// TIA Portal V20 export
FUNCTION_BLOCK "CallUnit"   // FB7, LAD
TITLE = CallUnit
AUTHOR : ERsystem_FA2_DH. Kim
// Unit logic and state machine
// stored: IsIECCheckEnabled true, MemoryReserve 100, Namespace Unit1, SetENOAutomatically false
   VAR_INPUT
      safetyReleased : Bool;   // Status from safety program
   END_VAR
   VAR_OUTPUT
      acknowledgeSafety { ExternalWritable := 'False'} : Bool;   // Acknowledge command to the safety program
   END_VAR
   VAR_IN_OUT
      globalStatus : "LAF_typeGeneralStatus";   // Global status
      unitInterface : "LAF_typeUnitInterface";   // Global unit interface
   END_VAR
   VAR
      instManageAlarms { ExternalWritable := 'False'} : "LAF_ManageAlarms";
      instStatusCollector { ExternalWritable := 'False'} : "LUC_StatusCollector";
      instInterfaceManager { ExternalWritable := 'False'} : "LUC_InterfaceManager";
      instUnitModeStateManager { ExternalWritable := 'False'} : "LPMLV2022_UnitModeStateManager";
      instRemoteInterfaceOpcUa { ExternalWritable := 'False'} : "LUC_RemoteCtrl_OpcUa";
      instSignalStack { ExternalWritable := 'False'} : "LUC_SignalStack";
      instUnitModeStateTimes { ExternalWritable := 'False'} : "LPMLV2022_UnitModeStateTimes";
      instUnitModeChangeAllowed { ExternalWritable := 'False'} : "LPMLV2022_UnitModeChangeAllowed";
      instPFEEvents { S7_SetPoint := 'True'} : "Unit1.EventsPFE";
      statTonTime { S7_SetPoint := 'True'} : Array[0..99] of TON_TIME;
      instTofTimer { ExternalWritable := 'False'} : Array[0..9] of TOF_TIME;
      instEQP_Interface_BA010 { ExternalWritable := 'False'} : "LER_EQP_Interface_ReelCut";
      instEQP_Interface_BA015 { ExternalWritable := 'False'} : "LER_EQP_Interface_ReelCut";
      instEQP_Interface_BA060 { ExternalWritable := 'False'} : "LER_EQP_Interface_Inspection";
      instEQP_Interface_BA030 { ExternalWritable := 'False'} : "LER_EQP_Interface_OtherStack";
      BSEND_Instance_BA10 { S7_SetPoint := 'True'} : BSEND;
      BRCV_Instance_BA10 { S7_SetPoint := 'True'} : BRCV;
      BSEND_Instance_BA15 { S7_SetPoint := 'True'} : BSEND;
      BRCV_Instance_BA15 { S7_SetPoint := 'True'} : BRCV;
      BSEND_Instance_BA40 { S7_SetPoint := 'True'} : BSEND;
      BRCV_Instance_BA40 { S7_SetPoint := 'True'} : BRCV;
      BSEND_Instance_BA60 { S7_SetPoint := 'True'} : BSEND;
      BRCV_Instance_BA60 { S7_SetPoint := 'True'} : BRCV;
      instSinaInfeed { ExternalWritable := 'False'} : SinaInfeed;
      statRemoteInterface { ExternalWritable := 'False'} : "LUC_typeCommands";
      statLocalInterface { ExternalWritable := 'False'} : "LUC_typeCommands";
      statEmEnableCheck { ExternalWritable := 'False'} : Array[0..2] of Bool;
      statSpecialFuctionEnableCheck : Array[0..2] of Bool;
      statEmHomeScCheck { ExternalWritable := 'False'} : Array[0..7] of Bool;
      statPulse { ExternalWritable := 'False'} : Array[0..99] of Bool;
      statNoModeCmd { ExternalWritable := 'False'} : Bool;
      statEnableManualCmds : Bool;
      sleep { S7_SetPoint := 'True'} : "LER_typeSleepMode";
      statPreElectrodeNumber : Struct
         anode : DInt;
         cathode : DInt;
         currentTotalEL : DInt;
      END_STRUCT;
      instCalculateOut { S7_SetPoint := 'True'} : "LER_Calculate_Out";
      instStackMainCommand { S7_SetPoint := 'True'} : "LER_StackMainCommand";
      InstLER_FFU_LIU117 { S7_SetPoint := 'True'} : "LER_FFU_LIU117";
      sMotionToPLC { S7_SetPoint := 'True'} : "LER_typeCommonDataStackMotion";
      StatAllEmLinked { S7_SetPoint := 'True'} : Bool;
      citi_Ptrig : Array[0..20] of Bool;
      citiTon : Array[0..20] of TON_TIME;
      citi : Time;
      citiTest : Array[0..20] of Bool;
      statCalculateParameters : Struct
         AnodeCount : DInt;
         CathodeCount : DInt;
         SepaCount : DInt;
         TotalThickness : LReal;
         TotalSepaWebLenth : LReal;
      END_STRUCT;
   END_VAR
   VAR_TEMP
      tempUnitFeedback : "LUC_typeEmFeedback";   // Collected commands in the unit, e.g. direct command or commands derived from alarms
      tempProcessCommands : "LUC_typeStateCommands";   // Requested unit state changes by the process
      tempUnitMode : DInt;   // Requested unit mode
      tempUnitModeChangeRequest : Bool;   // Request unit mode
      tempCntrlCmd : DInt;   // Request control command
      tempCmdChangeRequest : Bool;   // Enable change into requested state
      tempSc : Bool;   // State change from FALSE to TRUE (rising edge) triggers state complete signal
      tempFFuCount : Bool;
   END_VAR
   VAR CONSTANT
      TRUE : Bool := TRUE;
      FALSE : Bool := FALSE;
   END_VAR
   // // statLocalInterface.modeRequests.nomode : Request to change to "No Mode"
   // // statLocalInterface.modeRequests.sleep : Request to change to "Sleep Mode"
   // // statLocalInterface.modeRequests.deepsleep : Request to change to "Deep Sleep Mode"
   VAR_TEMP   // added for the SCL form of the ladder/FBD networks
      _w1 : Bool;
      _w2 : Bool;
      _w3 : Bool;
      _w4 : Bool;
      _w5 : Bool;
   END_VAR
BEGIN

REGION Network 1: BLOCK INFO HEADER
   // ERsystem / (C) Copyright 2025
   // ------------------------------------------------------------------------------
   // Title:            Call Unit
   // Comment/Function: Function to control unit mode and state transitions
   // Library/Family:   -
   // Author:           FA 2 / DH.Kim
   // Target System:    -
   // Engineering:      TIA Portal V20
   // Restrictions:     -
   // Requirements:     -
   // ------------------------------------------------------------------------------
   // Change log table:
   // Version     | Date       | Expert in charge | Changes applied ------------|------------|------------------|---------------------------------
   // 001.000.000 | 2025-03-29 | DH.Kim
   //                            First released version
END_REGION

REGION Network 2: DESCRIPTION
   // This function block is based on a template block provided by the Automation Framework.
   // It is used to control a unit structured according to the ISA-88 standard, and manages unit mode and state transitions in compliance with PackML.
   // 
   // - Mode changes can be triggered via HMI commands.
   // 
   // - State transitions are controlled either by feedback signals from equipment modules (EMs) or by HMI commands.
   // 
   // Additionally, this block handles feedback from DC24V and pneumatic sources, which is an exception to standard state transition logic.
END_REGION

REGION Network 3: Simulation
   // If simulation is active on a global level, inherit this status and set simulation active in this unit also. Information is written to DB ControlNodes, from where it is distributed to the equipmemt modules.
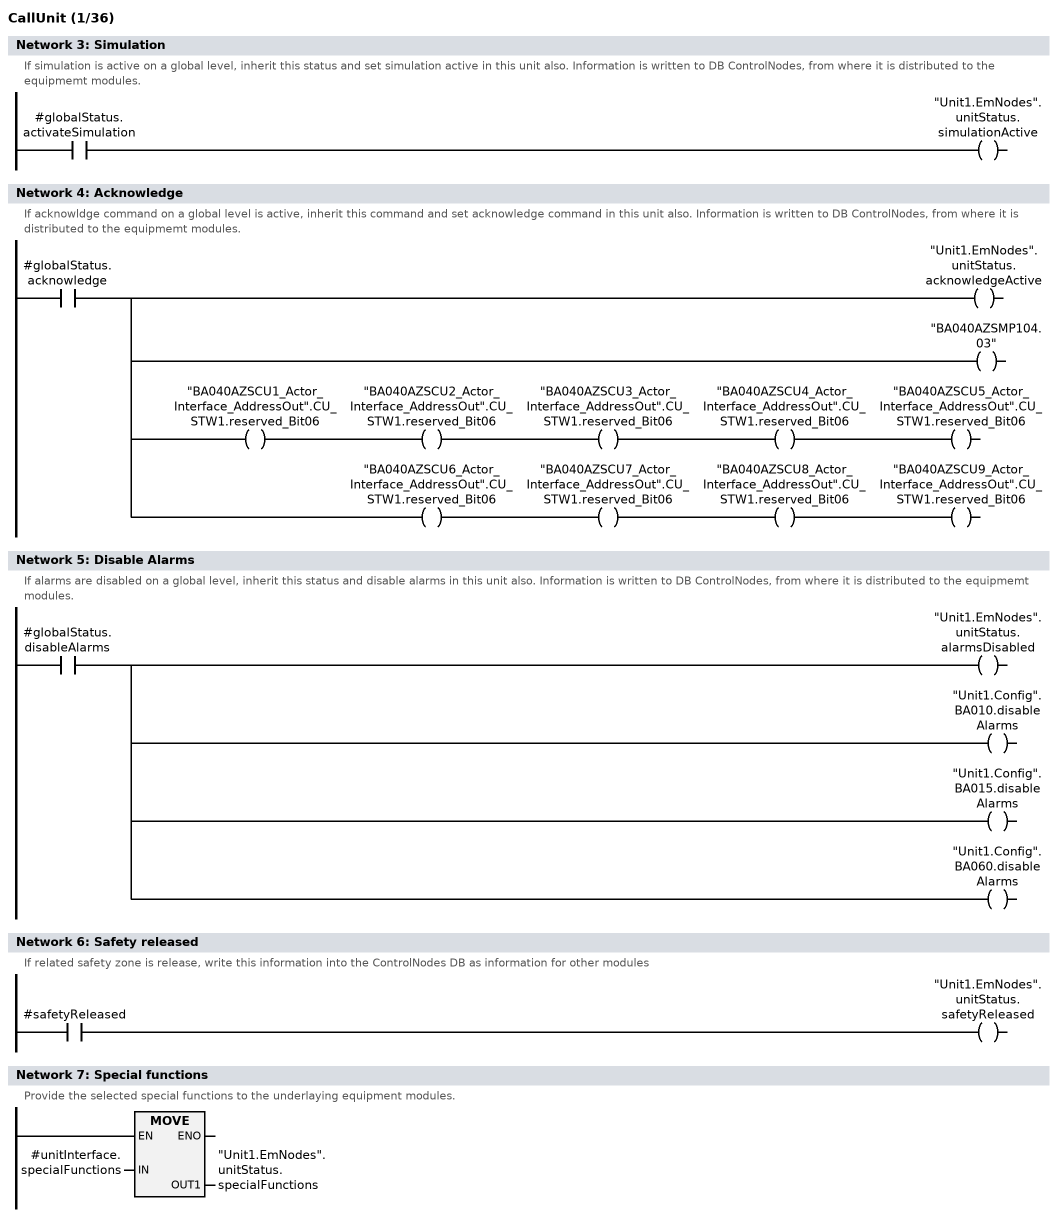
   RUNG wire#powerrail
      Contact( #globalStatus.activateSimulation )
      Coil( "Unit1.EmNodes".unitStatus.simulationActive )
   END_RUNG
   // the same network as SCL:
   "Unit1.EmNodes".unitStatus.simulationActive := #globalStatus.activateSimulation;
END_REGION

REGION Network 4: Acknowledge
   // If acknowldge command on a global level is active, inherit this command and set acknowledge command in this unit also. Information is written to DB ControlNodes, from where it is distributed to the equipmemt modules.
   RUNG wire#powerrail
      Contact( #globalStatus.acknowledge )
      wire#w1
      Coil( "Unit1.EmNodes".unitStatus.acknowledgeActive )
   END_RUNG
   RUNG wire#w1
      Coil( "BA040AZSMP104.03" )
   END_RUNG
   RUNG wire#w1
      Coil( "BA040AZSCU1_Actor_Interface_AddressOut".CU_STW1.reserved_Bit06 )
      Coil( "BA040AZSCU2_Actor_Interface_AddressOut".CU_STW1.reserved_Bit06 )
      Coil( "BA040AZSCU3_Actor_Interface_AddressOut".CU_STW1.reserved_Bit06 )
      Coil( "BA040AZSCU4_Actor_Interface_AddressOut".CU_STW1.reserved_Bit06 )
      Coil( "BA040AZSCU5_Actor_Interface_AddressOut".CU_STW1.reserved_Bit06 )
   END_RUNG
   RUNG wire#w1
      Coil( "BA040AZSCU6_Actor_Interface_AddressOut".CU_STW1.reserved_Bit06 )
      Coil( "BA040AZSCU7_Actor_Interface_AddressOut".CU_STW1.reserved_Bit06 )
      Coil( "BA040AZSCU8_Actor_Interface_AddressOut".CU_STW1.reserved_Bit06 )
      Coil( "BA040AZSCU9_Actor_Interface_AddressOut".CU_STW1.reserved_Bit06 )
   END_RUNG
   // the same network as SCL:
   "Unit1.EmNodes".unitStatus.acknowledgeActive := #globalStatus.acknowledge;
   "BA040AZSMP104.03" := #globalStatus.acknowledge;
   "BA040AZSCU1_Actor_Interface_AddressOut".CU_STW1.reserved_Bit06 := #globalStatus.acknowledge;
   "BA040AZSCU2_Actor_Interface_AddressOut".CU_STW1.reserved_Bit06 := #globalStatus.acknowledge;
   "BA040AZSCU3_Actor_Interface_AddressOut".CU_STW1.reserved_Bit06 := #globalStatus.acknowledge;
   "BA040AZSCU4_Actor_Interface_AddressOut".CU_STW1.reserved_Bit06 := #globalStatus.acknowledge;
   "BA040AZSCU5_Actor_Interface_AddressOut".CU_STW1.reserved_Bit06 := #globalStatus.acknowledge;
   "BA040AZSCU6_Actor_Interface_AddressOut".CU_STW1.reserved_Bit06 := #globalStatus.acknowledge;
   "BA040AZSCU7_Actor_Interface_AddressOut".CU_STW1.reserved_Bit06 := #globalStatus.acknowledge;
   "BA040AZSCU8_Actor_Interface_AddressOut".CU_STW1.reserved_Bit06 := #globalStatus.acknowledge;
   "BA040AZSCU9_Actor_Interface_AddressOut".CU_STW1.reserved_Bit06 := #globalStatus.acknowledge;
END_REGION

REGION Network 5: Disable Alarms
   // If alarms are disabled on a global level, inherit this status and disable alarms in this unit also. Information is written to DB ControlNodes, from where it is distributed to the equipmemt modules.
   RUNG wire#powerrail
      Contact( #globalStatus.disableAlarms )
      wire#w1
      Coil( "Unit1.EmNodes".unitStatus.alarmsDisabled )
   END_RUNG
   RUNG wire#w1
      Coil( "Unit1.Config".BA010.disableAlarms )
   END_RUNG
   RUNG wire#w1
      Coil( "Unit1.Config".BA015.disableAlarms )
   END_RUNG
   RUNG wire#w1
      Coil( "Unit1.Config".BA060.disableAlarms )
   END_RUNG
   // the same network as SCL:
   "Unit1.EmNodes".unitStatus.alarmsDisabled := #globalStatus.disableAlarms;
   "Unit1.Config".BA010.disableAlarms := #globalStatus.disableAlarms;
   "Unit1.Config".BA015.disableAlarms := #globalStatus.disableAlarms;
   "Unit1.Config".BA060.disableAlarms := #globalStatus.disableAlarms;
END_REGION

REGION Network 6: Safety released
   // If related safety zone is release, write this information into the ControlNodes DB as information for other modules
   RUNG wire#powerrail
      Contact( #safetyReleased )
      Coil( "Unit1.EmNodes".unitStatus.safetyReleased )
   END_RUNG
   // the same network as SCL:
   "Unit1.EmNodes".unitStatus.safetyReleased := #safetyReleased;
END_REGION

REGION Network 7: Special functions
   // Provide the selected special functions to the underlaying equipment modules.
   RUNG wire#powerrail
      Move(in := #unitInterface.specialFunctions, out1 => "Unit1.EmNodes".unitStatus.specialFunctions)
   END_RUNG
   // the same network as SCL:
   "Unit1.EmNodes".unitStatus.specialFunctions := #unitInterface.specialFunctions;
END_REGION

REGION Network 8 (SCL): Electric Power CB
   "Unit1.ControlNodes".fuses.motorpower_mcFeedBack := "BA040AZSCU1_Actor_Interface_AddressIn".E_DIGITAL.digitalInput0; //I5002.0
   "Unit1.ControlNodes".fuses.E202CB_motorpower_tripped := "BA040AZSCU1_Actor_Interface_AddressIn".E_DIGITAL.digitalInput1; //I5002.1
   "Unit1.ControlNodes".fuses.E208CB_maincontrol_panelMain_power_tripped := "BA040AZSCU1_Actor_Interface_AddressIn".E_DIGITAL.digitalInput2; //I5002.2
   "Unit1.ControlNodes".fuses.E320CB_E9304PWS_controlpower_SMPS_AC_power_tripped := "BA040AZSCU1_Actor_Interface_AddressIn".E_DIGITAL.digitalInput3; //I5002.3
   "Unit1.ControlNodes".fuses.E326CB_E9404PWS_controlpower_SMPS_AC_power_tripped := "BA040AZSCU1_Actor_Interface_AddressIn".E_DIGITAL.digitalInput4; //I5002.4
   "Unit1.ControlNodes".fuses.E400CB_compensator_X_Axis_power_TR_primarytripped := "BA040AZSCU1_Actor_Interface_AddressIn".E_DIGITAL.digitalInput6; //I5002.6
   "Unit1.ControlNodes".fuses.E410CB_compensator_X_Axis_power_TR_ECONDARYtripped := "BA040AZSCU1_Actor_Interface_AddressIn".E_DIGITAL.digitalInput7; //I5002.7

   "Unit1.ControlNodes".fuses.E500CB_sepa_pnp_X_Axis_powerTr_primary_tripped := "BA040AZSCU2_Actor_Interface_AddressIn".E_DIGITAL.digitalInput0; //I5006.0
   "Unit1.ControlNodes".fuses.E510CB_sepa_pnp_X_Axis_powerTr_ECONDARY_tripped := "BA040AZSCU2_Actor_Interface_AddressIn".E_DIGITAL.digitalInput1; //I5006.1
   "Unit1.ControlNodes".fuses.E720CB_powerMetrt_powerTRIIPED := "BA040AZSCU2_Actor_Interface_AddressIn".E_DIGITAL.digitalInput4; //I5006.4
   "Unit1.ControlNodes".fuses.E726CB_powerMetrt_controlpower_TRIIPED := "BA040AZSCU2_Actor_Interface_AddressIn".E_DIGITAL.digitalInput5; //I5006.5
   "Unit1.ControlNodes".fuses.E3304CB_compensator_X_Axis_power_onTrippred := "BA040AZSCU2_Actor_Interface_AddressIn".E_DIGITAL.digitalInput6; //I5006.6

   "Unit1.ControlNodes".fuses.E3504CB_sepa_pnp1_X_Axis_power_onTrippred := "BA040AZSCU3_Actor_Interface_AddressIn".E_DIGITAL.digitalInput0; //I5010.0
   "Unit1.ControlNodes".fuses.E3604CB_sepa_pnp2_X_Axis_power_onTrippred := "BA040AZSCU3_Actor_Interface_AddressIn".E_DIGITAL.digitalInput1; //I5010.1
   "Unit1.ControlNodes".fuses.E7116CB_procrssor_power_ontrippred := "BA040AZSCU3_Actor_Interface_AddressIn".E_DIGITAL.digitalInput4; //I5010.4
   "Unit1.ControlNodes".fuses.E7156CB_maincontrol_panelHot_power_tripped := "BA040AZSCU3_Actor_Interface_AddressIn".E_DIGITAL.digitalInput5; //I5010.5
   "Unit1.ControlNodes".fuses.E7304CB_panelLed_power_tripped := "BA040AZSCU3_Actor_Interface_AddressIn".E_DIGITAL.digitalInput6; //I5010.6

   "Unit1.ControlNodes".fuses.E8100CB_120VAC_control_powerTr_primary_tripped := "BA040AZSCU4_Actor_Interface_AddressIn".E_DIGITAL.digitalInput0; //I5014.0
   "Unit1.ControlNodes".fuses.E8110CB_120VAC_control_powerTr_secondary_tripped := "BA040AZSCU4_Actor_Interface_AddressIn".E_DIGITAL.digitalInput1; //I5014.1
   "Unit1.ControlNodes".fuses.E8116CB_control_power_ONtripped := "BA040AZSCU4_Actor_Interface_AddressIn".E_DIGITAL.digitalInput2; //I5014.2
   "Unit1.ControlNodes".fuses.E8156CB_maincontrol_panelControl_power_tripped := "BA040AZSCU4_Actor_Interface_AddressIn".E_DIGITAL.digitalInput3; //I5014.3
   "Unit1.ControlNodes".fuses.E9122CB_encoder_terminalUnit_control_power_tripped := "BA040AZSCU4_Actor_Interface_AddressIn".E_DIGITAL.digitalInput6; //I5014.6
   "Unit1.ControlNodes".fuses.E9128CB_servo_control_UNITcontrol_power_tripped := "BA040AZSCU4_Actor_Interface_AddressIn".E_DIGITAL.digitalInput7; //I5014.7

   "Unit1.ControlNodes".fuses.E9204CB_panelFan_power_tripped := "BA040AZSCU5_Actor_Interface_AddressIn".E_DIGITAL.digitalInput0; //I5018.0
   "Unit1.ControlNodes".fuses.E9306CB_controlDc_power_tripped := "BA040AZSCU5_Actor_Interface_AddressIn".E_DIGITAL.digitalInput2; //I5018.2
   "Unit1.ControlNodes".fuses.E9316CB_servo_control_power_tripped := "BA040AZSCU5_Actor_Interface_AddressIn".E_DIGITAL.digitalInput3; //I5018.3
   "Unit1.ControlNodes".fuses.E9406CB_controlDc_power_tripped := "BA040AZSCU5_Actor_Interface_AddressIn".E_DIGITAL.digitalInput5; //I5018.5
   "Unit1.ControlNodes".fuses.E9416CB_junctionBox_class_2SMPS_tripped := "BA040AZSCU5_Actor_Interface_AddressIn".E_DIGITAL.digitalInput6; //I5018.6
   "Unit1.ControlNodes".fuses.E9422CB_EQUIPMENT_LED_power_tripped := "BA040AZSCU5_Actor_Interface_AddressIn".E_DIGITAL.digitalInput7; //I5018.7

   "Unit1.ControlNodes".fuses.E214CB_E6404PWS_controlLER_power_SMPS_AC_power_tripped := "BA040AZSMP101.02";
   "Unit1.ControlNodes".fuses.E222CB_E6704PWS_controlLER_power_SMPS_AC_power_tripped := "BA040AZSMP101.03";
   "Unit1.ControlNodes".fuses.E226CB_E6804PWS_safety_power_SMPS_AC_power_tripped := "BA040AZSMP101.04";
   "Unit1.ControlNodes".fuses.E4120CB_procrssor_power_onTrpped := "BA040AZSMP101.06";
   "Unit1.ControlNodes".fuses.E4126CB_programing_power_outletTrpped := "BA040AZSMP101.07";
   "Unit1.ControlNodes".fuses.E4304CB_panelLed_power_tripped := "BA040AZSMP101.11";
   "Unit1.ControlNodes".fuses.E4420CB_controlLevel_hub_power_tripped := "BA040AZSMP101.14";
   "Unit1.ControlNodes".fuses.E4426CB_mainHmi_power_tripped := "BA040AZSMP101.15";
   "Unit1.ControlNodes".fuses.E4432CB_portableHmi_power_TIPPED := "BA040AZSMP101.16";
   "Unit1.ControlNodes".fuses.E4604CB_panelIrtHub_power_TIPPED := "BA040AZSMP101.17";
   "Unit1.ControlNodes".fuses.E4608ES_irtHub_fault := "BA040AZSMP101.20";
   "Unit1.ControlNodes".fuses.E5110CB_120VAC_control_power_TR_secondary_tripped := "BA040AZSMP101.23";
   "Unit1.ControlNodes".fuses.E5120CB_control_power_onTrippred := "BA040AZSMP101.24";
   "Unit1.ControlNodes".fuses.E5126CB_visionMonitor1_MCU_power_strip_outlet_power_tripped := "BA040AZSMP101.25";
   "Unit1.ControlNodes".fuses.E5132CB_visionMonitor2_visionMonitor3_power_strip_outlet_power_tripped := "BA040AZSMP101.26";
   "Unit1.ControlNodes".fuses.E5156CB_vision_LIGHT_controller_power_strip_outlet_power_tripped := #TRUE; //_."BA040AZSMP101.27";
   "Unit1.ControlNodes".fuses.E5222CB_FFU_power1_power_tripped := "BA040AZSMP101.31";
   "Unit1.ControlNodes".fuses.E6154CB_ET200MP_io_output_power_tripped := "BA040AZSMP101.34";
   "Unit1.ControlNodes".fuses.E6180CB_junctionBox_control_power_tripped := "BA040AZSMP101.35";
   "Unit1.ControlNodes".fuses.E6204CB_class2_SMPS_power_tripped := "BA040AZSMP101.36";
   "Unit1.ControlNodes".fuses.E6220CB_ET200ECO_PN1_power_tripped := "BA040AZSMP102.00";
   "Unit1.ControlNodes".fuses.E6224CB_ET200ECO_PN2_power_tripped := "BA040AZSMP102.01";
   "Unit1.ControlNodes".fuses.E6228CB_ET200ECO_PN3_power_tripped := "BA040AZSMP102.02";
   "Unit1.ControlNodes".fuses.E6232CB_ET200ECO_PN4_power_tripped := "BA040AZSMP102.03";
   "Unit1.ControlNodes".fuses.E6304CB_panelFan_power_tripped := "BA040AZSMP102.04";
   "Unit1.ControlNodes".fuses.E6406CB_controlLer_DC_power_tripped := "BA040AZSMP102.07";
   "Unit1.ControlNodes".fuses.E6422CB_mainFold1_control_power_tripped := "BA040AZSMP102.11";
   "Unit1.ControlNodes".fuses.E6430CB_mainFold2_control_power_tripped := "BA040AZSMP102.12";
   "Unit1.ControlNodes".fuses.E6456CB_driveCliq_hub_power_tripped := "BA040AZSMP102.13";
   "Unit1.ControlNodes".fuses.E6462CB_driveCliq_hub_power_tripped := "BA040AZSMP102.14";
   "Unit1.ControlNodes".fuses.E6468CB_handy_qr_reader_power_tripped := "BA040AZSMP102.15";
   "Unit1.ControlNodes".fuses.E6474CB_vision_controller1_power_tripped := "BA040AZSMP102.16";
   "Unit1.ControlNodes".fuses.E6480CB_vision_controller2_power_tripped := "BA040AZSMP102.17";
   "Unit1.ControlNodes".fuses.E6486CB_vision_controller3_power_tripped := "BA040AZSMP102.20";
   "Unit1.ControlNodes".fuses.E6506CB_linedLaser_module1_power_tripped := "BA040AZSMP102.21";
   "Unit1.ControlNodes".fuses.E6512CB_linedLaser_module2_power_tripped := "BA040AZSMP102.22";
   "Unit1.ControlNodes".fuses.E6706CB_controlLER_DC_power_tripped := "BA040AZSMP102.25";
   "Unit1.ControlNodes".fuses.E6716CB_EPC_controller1_power_tripped := "BA040AZSMP102.26";
   "Unit1.ControlNodes".fuses.E6722CB_EPC_controller2_power_tripped := "BA040AZSMP102.27";
   "Unit1.ControlNodes".fuses.E6728CB_EPC_controller3_power_tripped := "BA040AZSMP102.30";
   "Unit1.ControlNodes".fuses.E6734CB_EPC_controller4_power_tripped := "BA040AZSMP102.31";
   "Unit1.ControlNodes".fuses.E6806CB_safetyDc_power_tripped := "BA040AZSMP102.33";
   "Unit1.ControlNodes".fuses.E6816CB_ET200SP_io_safety_power_tripped := "BA040AZSMP102.34";
   "Unit1.ControlNodes".fuses.E6836CB_junctionBox_control_power_tripped := "BA040AZSMP102.35";
   "Unit1.ControlNodes".fuses.E6856CB_ET200ECO_PN_safety_1_power_tripped := "BA040AZSMP102.36";
   "Unit1.ControlNodes".fuses.E6862CB_ET200ECO_PN_safety_2_power_tripped := "BA040AZSMP102.37";
   "Unit1.ControlNodes".fuses.E6756CB_dcdc_converter_in_power_tripped := "BA040AZSMP103.00";
   "Unit1.ControlNodes".fuses.E6762CB_hotWire_cutter_power_tripped := "BA040AZSMP103.01";
   "Unit1.ControlNodes".fuses.E110CB_mainHmi_power_tripped := "BA040AZSSP201.10";
END_REGION

REGION Network 9 (SCL): Power Supply
   "Unit1.ControlNodes".pws.E9104PWS_control_power_smpSdc_ok := "BA040AZSCU4_Actor_Interface_AddressIn".E_DIGITAL.digitalInput4; //I5014.4
   "Unit1.ControlNodes".pws.E9304PWS_control_power_smpSdc_ok := "BA040AZSCU5_Actor_Interface_AddressIn".E_DIGITAL.digitalInput1; //I5018.1
   "Unit1.ControlNodes".pws.E9404PWS_control_power_smpSdc_ok := "BA040AZSCU5_Actor_Interface_AddressIn".E_DIGITAL.digitalInput4; //I5018.4

   "Unit1.ControlNodes".pws.E4404PWS_plc_powerSmpsDc_ok := "BA040AZSMP101.13";
   "Unit1.ControlNodes".pws.E6104PWS_control_powerSmpsDc_ok := "BA040AZSMP101.33";
   "Unit1.ControlNodes".pws.E6206PWS_class2_smps_monitoring := "BA040AZSMP101.37";
   "Unit1.ControlNodes".pws.E6404PWS_controller_powerSmpsDc_ok := "BA040AZSMP102.06";
   "Unit1.ControlNodes".pws.E6704PWS_controller_powerSmpsDc_ok := "BA040AZSMP102.24";
   "Unit1.ControlNodes".pws.E6804PWS_safety_powerSmpsDc_ok := "BA040AZSMP102.32";
END_REGION

REGION Network 10: Main Air Ok
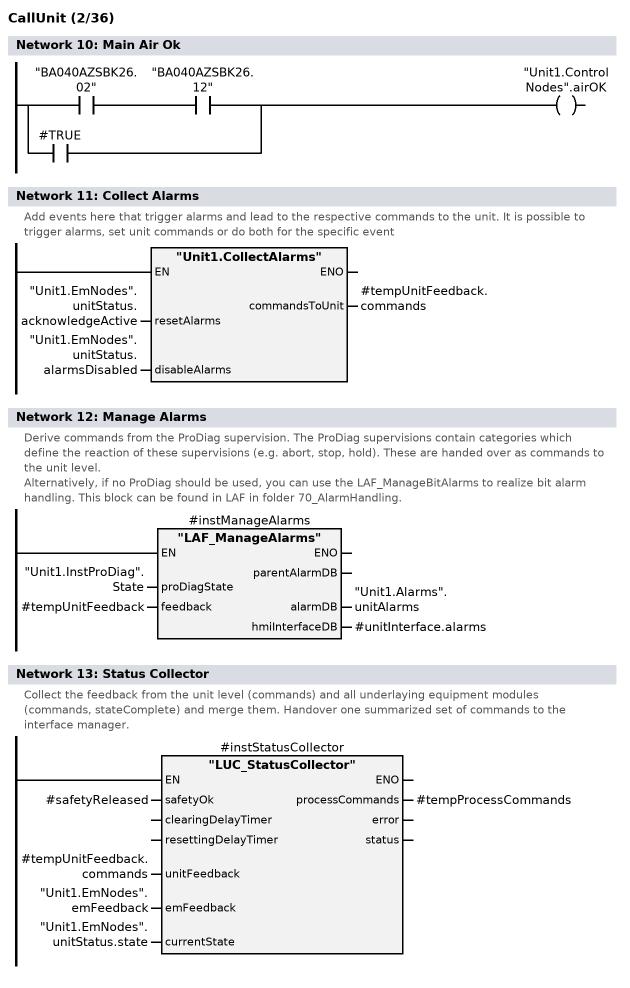
   RUNG wire#powerrail
      Contact( "BA040AZSBK26.02" )
      Contact( "BA040AZSBK26.12" )
      wire#w1
      Coil( "Unit1.ControlNodes".airOK )
   END_RUNG
   RUNG wire#powerrail
      Contact( #TRUE )
   END_RUNG wire#w1
   // the same network as SCL:
   "Unit1.ControlNodes".airOK := ("BA040AZSBK26.02" AND "BA040AZSBK26.12") OR #TRUE;
END_REGION

REGION Network 11: Collect Alarms
   // Add events here that trigger alarms and lead to the respective commands to the unit. It is possible to trigger alarms, set unit commands or do both for the specific event
   RUNG wire#powerrail
      "Unit1.CollectAlarms"(resetAlarms := "Unit1.EmNodes".unitStatus.acknowledgeActive, disableAlarms := "Unit1.EmNodes".unitStatus.alarmsDisabled, commandsToUnit => #tempUnitFeedback.commands)
   END_RUNG
   // the same network as SCL:
   "Unit1.CollectAlarms"(resetAlarms := "Unit1.EmNodes".unitStatus.acknowledgeActive,
                         disableAlarms := "Unit1.EmNodes".unitStatus.alarmsDisabled,
                         commandsToUnit => #tempUnitFeedback.commands);
END_REGION

REGION Network 12: Manage Alarms
   // Derive commands from the ProDiag supervision. The ProDiag supervisions contain categories which define the reaction of these supervisions (e.g. abort, stop, hold). These are handed over as commands to the unit level.
   // Alternatively, if no ProDiag should be used, you can use the LAF_ManageBitAlarms to realize bit alarm handling. This block can be found in LAF in folder 70_AlarmHandling.
   RUNG wire#powerrail
      #instManageAlarms(proDiagState := "Unit1.InstProDiag".State, feedback := #tempUnitFeedback, parentAlarmDB =>, alarmDB => "Unit1.Alarms".unitAlarms, hmiInterfaceDB => #unitInterface.alarms)
   END_RUNG
   // the same network as SCL:
   #instManageAlarms(proDiagState := "Unit1.InstProDiag".State,   // "LAF_ManageAlarms"
                     feedback := #tempUnitFeedback,
                     alarmDB => "Unit1.Alarms".unitAlarms,
                     hmiInterfaceDB => #unitInterface.alarms);
END_REGION

REGION Network 13: Status Collector
   // Collect the feedback from the unit level (commands) and all underlaying equipment modules (commands, stateComplete) and merge them. Handover one summarized set of commands to the interface manager.
   RUNG wire#powerrail
      #instStatusCollector(safetyOk := #safetyReleased, clearingDelayTimer :=, resettingDelayTimer :=, unitFeedback := #tempUnitFeedback.commands, emFeedback := "Unit1.EmNodes".emFeedback, currentState := "Unit1.EmNodes".unitStatus.state, processCommands => #tempProcessCommands, error =>, status =>)
   END_RUNG
   // the same network as SCL:
   #instStatusCollector(safetyOk := #safetyReleased,   // "LUC_StatusCollector"
                        unitFeedback := #tempUnitFeedback.commands,
                        emFeedback := "Unit1.EmNodes".emFeedback,
                        currentState := "Unit1.EmNodes".unitStatus.state,
                        processCommands => #tempProcessCommands);
END_REGION

REGION Network 14: Interface Manager
   // Read the commands from all interfaces (process, local, hmi, remote) and merge them. Handover one summarized set of commands to the mode state manager.
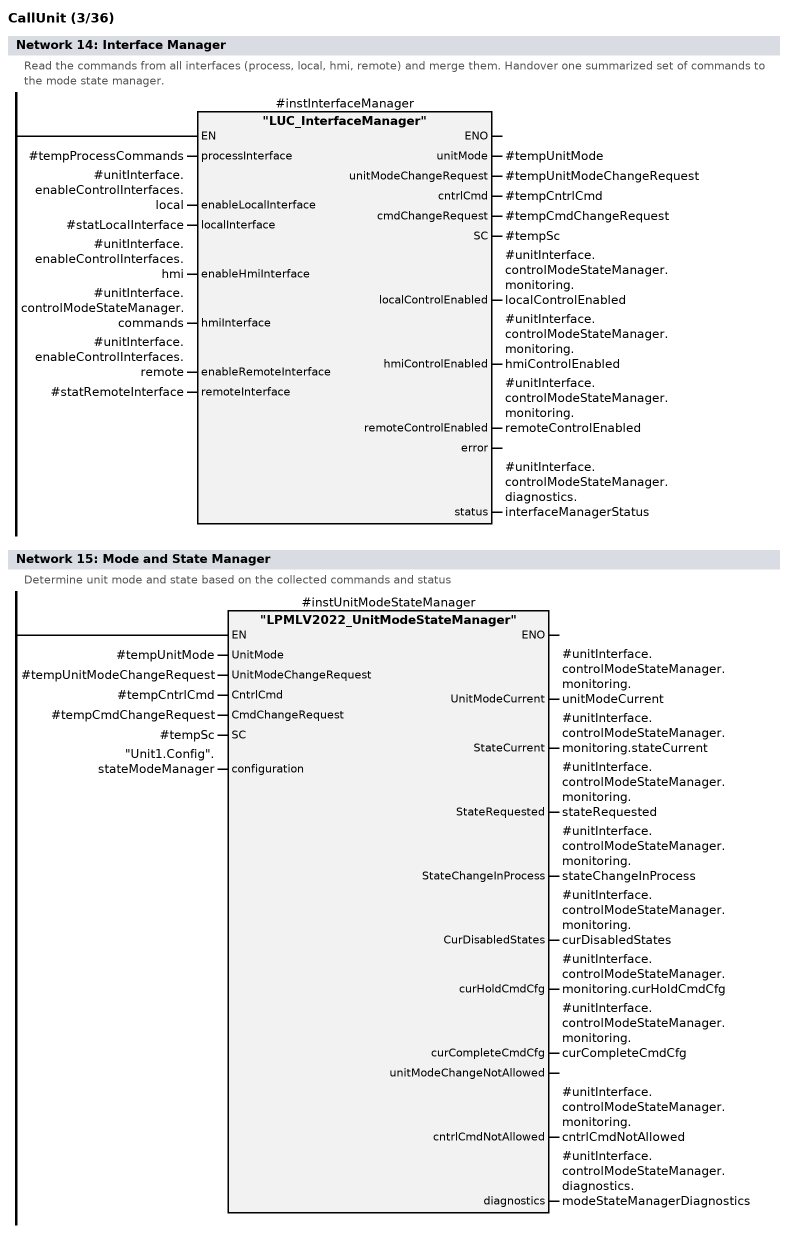
   RUNG wire#powerrail
      #instInterfaceManager(processInterface := #tempProcessCommands, enableLocalInterface := #unitInterface.enableControlInterfaces.local, localInterface := #statLocalInterface, enableHmiInterface := #unitInterface.enableControlInterfaces.hmi, hmiInterface := #unitInterface.controlModeStateManager.commands, enableRemoteInterface := #unitInterface.enableControlInterfaces.remote, remoteInterface := #statRemoteInterface, unitMode => #tempUnitMode, unitModeChangeRequest => #tempUnitModeChangeRequest, cntrlCmd => #tempCntrlCmd, cmdChangeRequest => #tempCmdChangeRequest, SC => #tempSc, localControlEnabled => #unitInterface.controlModeStateManager.monitoring.localControlEnabled, hmiControlEnabled => #unitInterface.controlModeStateManager.monitoring.hmiControlEnabled, remoteControlEnabled => #unitInterface.controlModeStateManager.monitoring.remoteControlEnabled, error =>, status => #unitInterface.controlModeStateManager.diagnostics.interfaceManagerStatus)
   END_RUNG
   // the same network as SCL:
   #instInterfaceManager(processInterface := #tempProcessCommands,   // "LUC_InterfaceManager"
                         enableLocalInterface := #unitInterface.enableControlInterfaces.local,
                         localInterface := #statLocalInterface,
                         enableHmiInterface := #unitInterface.enableControlInterfaces.hmi,
                         hmiInterface := #unitInterface.controlModeStateManager.commands,
                         enableRemoteInterface := #unitInterface.enableControlInterfaces.remote,
                         remoteInterface := #statRemoteInterface,
                         unitMode => #tempUnitMode,
                         unitModeChangeRequest => #tempUnitModeChangeRequest,
                         cntrlCmd => #tempCntrlCmd,
                         cmdChangeRequest => #tempCmdChangeRequest,
                         SC => #tempSc,
                         localControlEnabled => #unitInterface.controlModeStateManager.monitoring.localControlEnabled,
                         hmiControlEnabled => #unitInterface.controlModeStateManager.monitoring.hmiControlEnabled,
                         remoteControlEnabled => #unitInterface.controlModeStateManager.monitoring.remoteControlEnabled,
                         status => #unitInterface.controlModeStateManager.diagnostics.interfaceManagerStatus);
END_REGION

REGION Network 15: Mode and State Manager
   // Determine unit mode and state based on the collected commands and status
   RUNG wire#powerrail
      #instUnitModeStateManager(UnitMode := #tempUnitMode, UnitModeChangeRequest := #tempUnitModeChangeRequest, CntrlCmd := #tempCntrlCmd, CmdChangeRequest := #tempCmdChangeRequest, SC := #tempSc, configuration := "Unit1.Config".stateModeManager, UnitModeCurrent => #unitInterface.controlModeStateManager.monitoring.unitModeCurrent, StateCurrent => #unitInterface.controlModeStateManager.monitoring.stateCurrent, StateRequested => #unitInterface.controlModeStateManager.monitoring.stateRequested, StateChangeInProcess => #unitInterface.controlModeStateManager.monitoring.stateChangeInProcess, CurDisabledStates => #unitInterface.controlModeStateManager.monitoring.curDisabledStates, curHoldCmdCfg => #unitInterface.controlModeStateManager.monitoring.curHoldCmdCfg, curCompleteCmdCfg => #unitInterface.controlModeStateManager.monitoring.curCompleteCmdCfg, unitModeChangeNotAllowed =>, cntrlCmdNotAllowed => #unitInterface.controlModeStateManager.monitoring.cntrlCmdNotAllowed, diagnostics => #unitInterface.controlModeStateManager.diagnostics.modeStateManagerDiagnostics)
   END_RUNG
   // the same network as SCL:
   #instUnitModeStateManager(UnitMode := #tempUnitMode,   // "LPMLV2022_UnitModeStateManager"
                           UnitModeChangeRequest := #tempUnitModeChangeRequest,
                           CntrlCmd := #tempCntrlCmd,
                           CmdChangeRequest := #tempCmdChangeRequest,
                           SC := #tempSc,
                           configuration := "Unit1.Config".stateModeManager,
                           UnitModeCurrent => #unitInterface.controlModeStateManager.monitoring.unitModeCurrent,
                           StateCurrent => #unitInterface.controlModeStateManager.monitoring.stateCurrent,
                           StateRequested => #unitInterface.controlModeStateManager.monitoring.stateRequested,
                           StateChangeInProcess => #unitInterface.controlModeStateManager.monitoring.stateChangeInProcess,
                           CurDisabledStates => #unitInterface.controlModeStateManager.monitoring.curDisabledStates,
                           curHoldCmdCfg => #unitInterface.controlModeStateManager.monitoring.curHoldCmdCfg,
                           curCompleteCmdCfg => #unitInterface.controlModeStateManager.monitoring.curCompleteCmdCfg,
                           cntrlCmdNotAllowed => #unitInterface.controlModeStateManager.monitoring.cntrlCmdNotAllowed,
                           diagnostics => #unitInterface.controlModeStateManager.diagnostics.modeStateManagerDiagnostics);
END_REGION

REGION Network 16: Helper Functions
   // 1. Read mode and state from the mode state manager an write them to the DB ControlNode
   // 2. Read mode and state from the mode state manager, translate them to a string and write them in unitInterface
   // 3. Determine if a mode change is allowed in the current state and write that information to the unitInterface
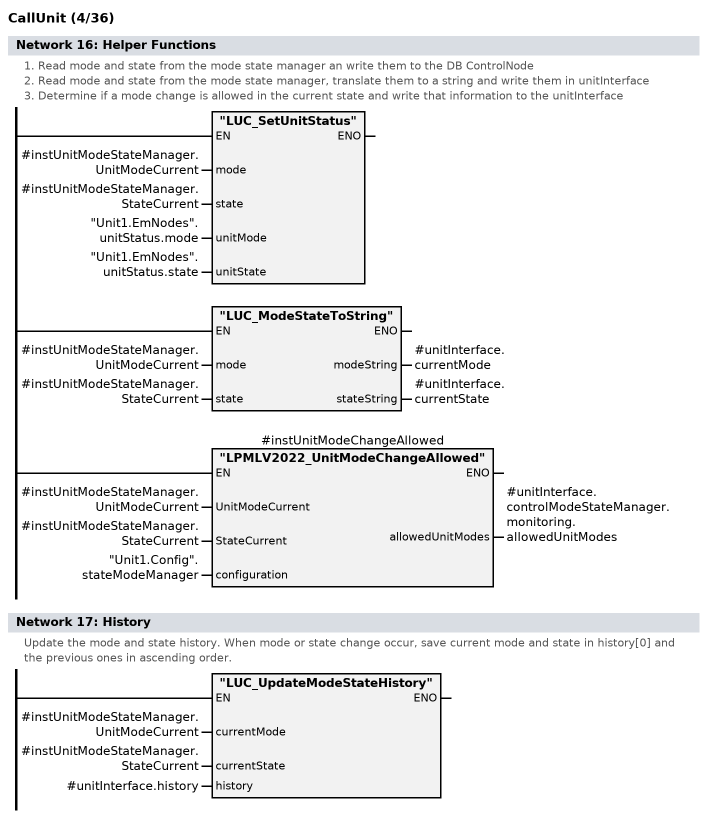
   RUNG wire#powerrail
      "LUC_SetUnitStatus"(mode := #instUnitModeStateManager.UnitModeCurrent, state := #instUnitModeStateManager.StateCurrent, unitMode := "Unit1.EmNodes".unitStatus.mode, unitState := "Unit1.EmNodes".unitStatus.state)
   END_RUNG
   RUNG wire#powerrail
      "LUC_ModeStateToString"(mode := #instUnitModeStateManager.UnitModeCurrent, state := #instUnitModeStateManager.StateCurrent, modeString => #unitInterface.currentMode, stateString => #unitInterface.currentState)
   END_RUNG
   RUNG wire#powerrail
      #instUnitModeChangeAllowed(UnitModeCurrent := #instUnitModeStateManager.UnitModeCurrent, StateCurrent := #instUnitModeStateManager.StateCurrent, configuration := "Unit1.Config".stateModeManager, allowedUnitModes => #unitInterface.controlModeStateManager.monitoring.allowedUnitModes)
   END_RUNG
   // the same network as SCL:
   "LUC_SetUnitStatus"(mode := #instUnitModeStateManager.UnitModeCurrent,
                       state := #instUnitModeStateManager.StateCurrent,
                       unitMode := "Unit1.EmNodes".unitStatus.mode,
                       unitState := "Unit1.EmNodes".unitStatus.state);
   "LUC_ModeStateToString"(mode := #instUnitModeStateManager.UnitModeCurrent,
                           state := #instUnitModeStateManager.StateCurrent,
                           modeString => #unitInterface.currentMode,
                           stateString => #unitInterface.currentState);
   #instUnitModeChangeAllowed(UnitModeCurrent := #instUnitModeStateManager.UnitModeCurrent,   // "LPMLV2022_UnitModeChangeAllowed"
                           StateCurrent := #instUnitModeStateManager.StateCurrent,
                           configuration := "Unit1.Config".stateModeManager,
                           allowedUnitModes => #unitInterface.controlModeStateManager.monitoring.allowedUnitModes);
END_REGION

REGION Network 17: History
   // Update the mode and state history. When mode or state change occur, save current mode and state in history[0] and the previous ones in ascending order.
   RUNG wire#powerrail
      "LUC_UpdateModeStateHistory"(currentMode := #instUnitModeStateManager.UnitModeCurrent, currentState := #instUnitModeStateManager.StateCurrent, history := #unitInterface.history)
   END_RUNG
   // the same network as SCL:
   "LUC_UpdateModeStateHistory"(currentMode := #instUnitModeStateManager.UnitModeCurrent,
                           currentState := #instUnitModeStateManager.StateCurrent,
                           history := #unitInterface.history);
END_REGION

REGION Network 18: Time Statistics
   // Determine the time that has been spend in modes and states.
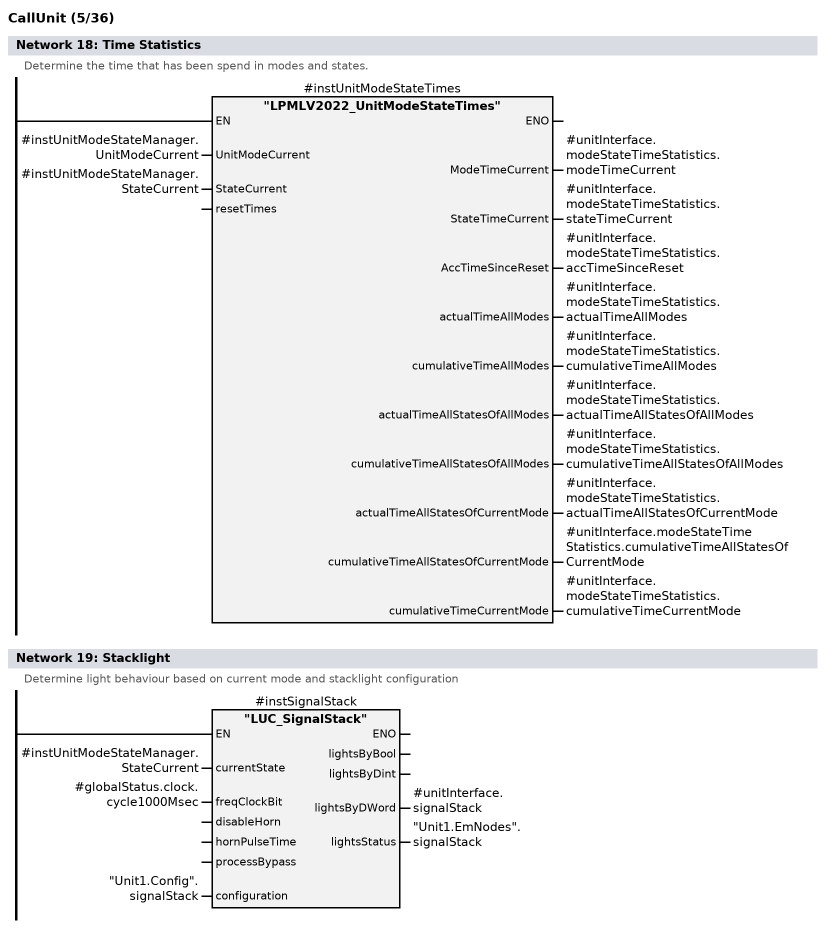
   RUNG wire#powerrail
      #instUnitModeStateTimes(UnitModeCurrent := #instUnitModeStateManager.UnitModeCurrent, StateCurrent := #instUnitModeStateManager.StateCurrent, resetTimes :=, ModeTimeCurrent => #unitInterface.modeStateTimeStatistics.modeTimeCurrent, StateTimeCurrent => #unitInterface.modeStateTimeStatistics.stateTimeCurrent, AccTimeSinceReset => #unitInterface.modeStateTimeStatistics.accTimeSinceReset, actualTimeAllModes => #unitInterface.modeStateTimeStatistics.actualTimeAllModes, cumulativeTimeAllModes => #unitInterface.modeStateTimeStatistics.cumulativeTimeAllModes, actualTimeAllStatesOfAllModes => #unitInterface.modeStateTimeStatistics.actualTimeAllStatesOfAllModes, cumulativeTimeAllStatesOfAllModes => #unitInterface.modeStateTimeStatistics.cumulativeTimeAllStatesOfAllModes, actualTimeAllStatesOfCurrentMode => #unitInterface.modeStateTimeStatistics.actualTimeAllStatesOfCurrentMode, cumulativeTimeAllStatesOfCurrentMode => #unitInterface.modeStateTimeStatistics.cumulativeTimeAllStatesOfCurrentMode, cumulativeTimeCurrentMode => #unitInterface.modeStateTimeStatistics.cumulativeTimeCurrentMode)
   END_RUNG
   // the same network as SCL:
   #instUnitModeStateTimes(UnitModeCurrent := #instUnitModeStateManager.UnitModeCurrent,   // "LPMLV2022_UnitModeStateTimes"
                           StateCurrent := #instUnitModeStateManager.StateCurrent,
                           ModeTimeCurrent => #unitInterface.modeStateTimeStatistics.modeTimeCurrent,
                           StateTimeCurrent => #unitInterface.modeStateTimeStatistics.stateTimeCurrent,
                           AccTimeSinceReset => #unitInterface.modeStateTimeStatistics.accTimeSinceReset,
                           actualTimeAllModes => #unitInterface.modeStateTimeStatistics.actualTimeAllModes,
                           cumulativeTimeAllModes => #unitInterface.modeStateTimeStatistics.cumulativeTimeAllModes,
                           actualTimeAllStatesOfAllModes => #unitInterface.modeStateTimeStatistics.actualTimeAllStatesOfAllModes,
                           cumulativeTimeAllStatesOfAllModes => #unitInterface.modeStateTimeStatistics.cumulativeTimeAllStatesOfAllModes,
                           actualTimeAllStatesOfCurrentMode => #unitInterface.modeStateTimeStatistics.actualTimeAllStatesOfCurrentMode,
                           cumulativeTimeAllStatesOfCurrentMode => #unitInterface.modeStateTimeStatistics.cumulativeTimeAllStatesOfCurrentMode,
                           cumulativeTimeCurrentMode => #unitInterface.modeStateTimeStatistics.cumulativeTimeCurrentMode);
END_REGION

REGION Network 19: Stacklight
   // Determine light behaviour based on current mode and stacklight configuration
   RUNG wire#powerrail
      #instSignalStack(currentState := #instUnitModeStateManager.StateCurrent, freqClockBit := #globalStatus.clock.cycle1000Msec, disableHorn :=, hornPulseTime :=, processBypass :=, configuration := "Unit1.Config".signalStack, lightsByBool =>, lightsByDint =>, lightsByDWord => #unitInterface.signalStack, lightsStatus => "Unit1.EmNodes".signalStack)
   END_RUNG
   // the same network as SCL:
   #instSignalStack(currentState := #instUnitModeStateManager.StateCurrent,   // "LUC_SignalStack"
                    freqClockBit := #globalStatus.clock.cycle1000Msec,
                    configuration := "Unit1.Config".signalStack,
                    lightsByDWord => #unitInterface.signalStack,
                    lightsStatus => "Unit1.EmNodes".signalStack);
END_REGION

REGION Network 20: Remote Control via OPC UA
   // Control the mode state manager remotely via OPC UA
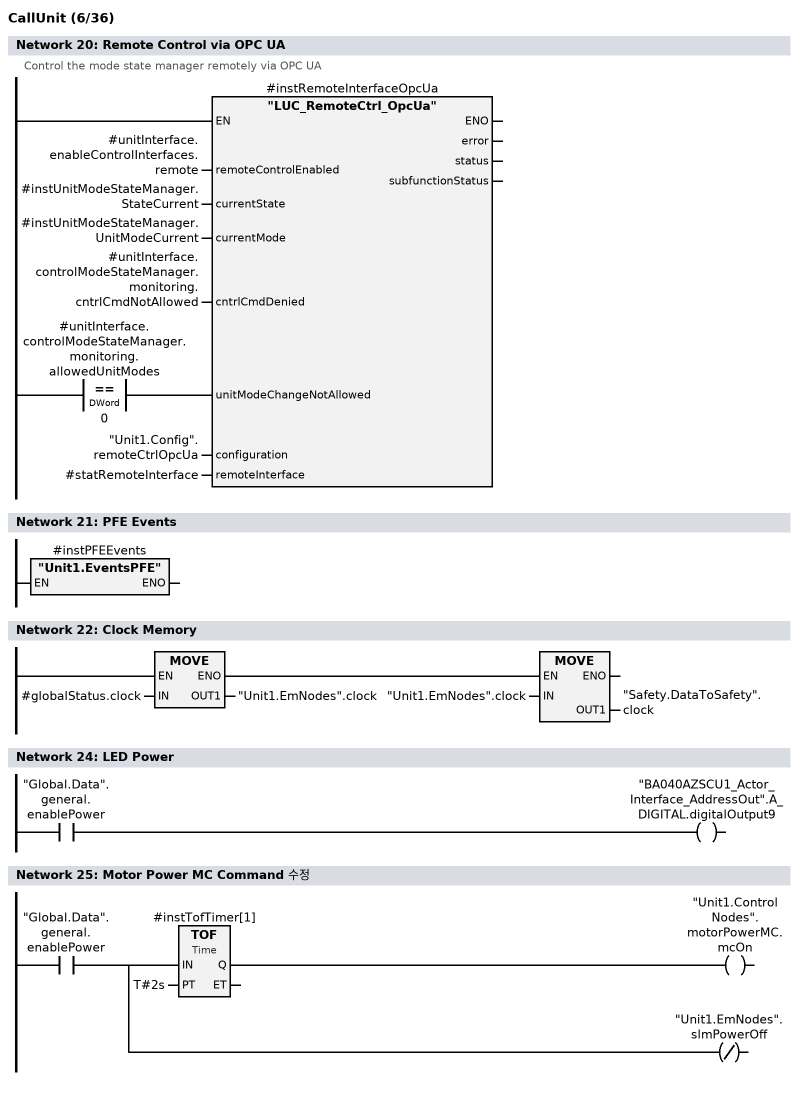
   RUNG wire#powerrail
      #instRemoteInterfaceOpcUa(unitModeChangeNotAllowed := wire#w1, remoteControlEnabled := #unitInterface.enableControlInterfaces.remote, currentState := #instUnitModeStateManager.StateCurrent, currentMode := #instUnitModeStateManager.UnitModeCurrent, cntrlCmdDenied := #unitInterface.controlModeStateManager.monitoring.cntrlCmdNotAllowed, configuration := "Unit1.Config".remoteCtrlOpcUa, remoteInterface := #statRemoteInterface, error =>, status =>, subfunctionStatus =>)
   END_RUNG
   RUNG wire#powerrail
      { S7_Templates := "SrcType := DWord" } EQ_Contact(in1 := #unitInterface.controlModeStateManager.monitoring.allowedUnitModes, in2 := 0)
   END_RUNG wire#w1
   // the same network as SCL:
   #instRemoteInterfaceOpcUa(remoteControlEnabled := #unitInterface.enableControlInterfaces.remote,   // "LUC_RemoteCtrl_OpcUa"
                           currentState := #instUnitModeStateManager.StateCurrent,
                           currentMode := #instUnitModeStateManager.UnitModeCurrent,
                           cntrlCmdDenied := #unitInterface.controlModeStateManager.monitoring.cntrlCmdNotAllowed,
                           unitModeChangeNotAllowed := #unitInterface.controlModeStateManager.monitoring.allowedUnitModes = 0,
                           configuration := "Unit1.Config".remoteCtrlOpcUa,
                           remoteInterface := #statRemoteInterface);
END_REGION

REGION Network 21: PFE Events
   RUNG wire#powerrail
      #instPFEEvents()
   END_RUNG
   // the same network as SCL:
   #instPFEEvents();   // "Unit1.EventsPFE"
END_REGION

REGION Network 22: Clock Memory
   RUNG wire#powerrail
      Move(in := #globalStatus.clock, out1 => "Unit1.EmNodes".clock)
      Move(in := "Unit1.EmNodes".clock, out1 => "Safety.DataToSafety".clock)
   END_RUNG
   // the same network as SCL:
   "Unit1.EmNodes".clock := #globalStatus.clock;
   "Safety.DataToSafety".clock := "Unit1.EmNodes".clock;
END_REGION

REGION Network 23: ******************** Power ********************
END_REGION

REGION Network 24: LED Power
   RUNG wire#powerrail
      Contact( "Global.Data".general.enablePower )
      Coil( "BA040AZSCU1_Actor_Interface_AddressOut".A_DIGITAL.digitalOutput9 )
   END_RUNG
   // the same network as SCL:
   "BA040AZSCU1_Actor_Interface_AddressOut".A_DIGITAL.digitalOutput9 := "Global.Data".general.enablePower;
END_REGION

REGION Network 25: Motor Power MC Command 수정
   RUNG wire#powerrail
      Contact( "Global.Data".general.enablePower )
      wire#w1
      { S7_Templates := "time_type := Time" } #instTofTimer[1].TOF(pt := T#2s, et =>)
      Coil( "Unit1.ControlNodes".motorPowerMC.mcOn )
   END_RUNG
   RUNG wire#w1
      I_Coil( "Unit1.EmNodes".slmPowerOff )
   END_RUNG
   // the same network as SCL:
   #instTofTimer[1].TOF(IN := "Global.Data".general.enablePower, PT := T#2s);
   "Unit1.ControlNodes".motorPowerMC.mcOn := #instTofTimer[1].Q;
   "Unit1.EmNodes".slmPowerOff := NOT "Global.Data".general.enablePower;
END_REGION

REGION Network 26: Motor Power MC Monitoring 수정
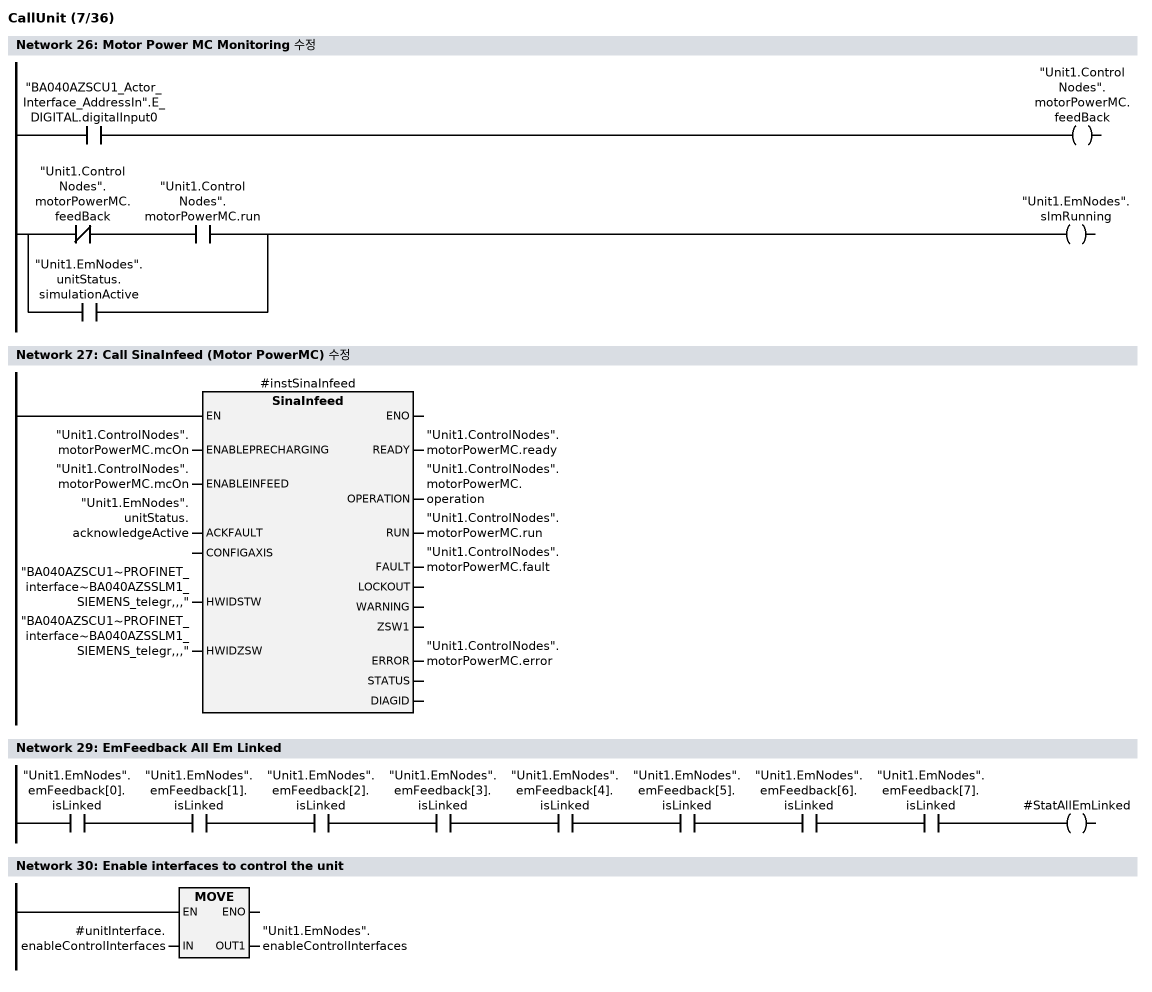
   RUNG wire#powerrail
      Contact( "BA040AZSCU1_Actor_Interface_AddressIn".E_DIGITAL.digitalInput0 )
      Coil( "Unit1.ControlNodes".motorPowerMC.feedBack )
   END_RUNG
   RUNG wire#powerrail
      I_Contact( "Unit1.ControlNodes".motorPowerMC.feedBack )
      Contact( "Unit1.ControlNodes".motorPowerMC.run )
      wire#w1
      Coil( "Unit1.EmNodes".slmRunning )
   END_RUNG
   RUNG wire#powerrail
      Contact( "Unit1.EmNodes".unitStatus.simulationActive )
   END_RUNG wire#w1
   // the same network as SCL:
   "Unit1.ControlNodes".motorPowerMC.feedBack := "BA040AZSCU1_Actor_Interface_AddressIn".E_DIGITAL.digitalInput0;
   "Unit1.EmNodes".slmRunning := (NOT "Unit1.ControlNodes".motorPowerMC.feedBack AND "Unit1.ControlNodes".motorPowerMC.run) OR "Unit1.EmNodes".unitStatus.simulationActive;
END_REGION

REGION Network 27: Call SinaInfeed (Motor PowerMC) 수정
   RUNG wire#powerrail
      #instSinaInfeed.SinaInfeed(EnablePrecharging := "Unit1.ControlNodes".motorPowerMC.mcOn, EnableInfeed := "Unit1.ControlNodes".motorPowerMC.mcOn, AckFault := "Unit1.EmNodes".unitStatus.acknowledgeActive, ConfigAxis :=, HWIDSTW := "BA040AZSCU1~PROFINET_interface~BA040AZSSLM1_SIEMENS_telegr,,,", HWIDZSW := "BA040AZSCU1~PROFINET_interface~BA040AZSSLM1_SIEMENS_telegr,,,", Ready => "Unit1.ControlNodes".motorPowerMC.ready, Operation => "Unit1.ControlNodes".motorPowerMC.operation, Run => "Unit1.ControlNodes".motorPowerMC.run, Fault => "Unit1.ControlNodes".motorPowerMC.fault, Lockout =>, Warning =>, ZSW1 =>, Error => "Unit1.ControlNodes".motorPowerMC.error, Status =>, DiagID =>)
   END_RUNG
   // the same network as SCL:
   #instSinaInfeed(EnablePrecharging := "Unit1.ControlNodes".motorPowerMC.mcOn,   // SinaInfeed
                   EnableInfeed := "Unit1.ControlNodes".motorPowerMC.mcOn,
                   AckFault := "Unit1.EmNodes".unitStatus.acknowledgeActive,
                   HWIDSTW := "BA040AZSCU1~PROFINET_interface~BA040AZSSLM1_SIEMENS_telegr,,,",
                   HWIDZSW := "BA040AZSCU1~PROFINET_interface~BA040AZSSLM1_SIEMENS_telegr,,,",
                   Ready => "Unit1.ControlNodes".motorPowerMC.ready,
                   Operation => "Unit1.ControlNodes".motorPowerMC.operation,
                   Run => "Unit1.ControlNodes".motorPowerMC.run,
                   Fault => "Unit1.ControlNodes".motorPowerMC.fault,
                   Error => "Unit1.ControlNodes".motorPowerMC.error);
END_REGION

REGION Network 28: ******************** Local Operation Box ********************
END_REGION

REGION Network 29: EmFeedback All Em Linked
   RUNG wire#powerrail
      Contact( "Unit1.EmNodes".emFeedback[0].isLinked )
      Contact( "Unit1.EmNodes".emFeedback[1].isLinked )
      Contact( "Unit1.EmNodes".emFeedback[2].isLinked )
      Contact( "Unit1.EmNodes".emFeedback[3].isLinked )
      Contact( "Unit1.EmNodes".emFeedback[4].isLinked )
      Contact( "Unit1.EmNodes".emFeedback[5].isLinked )
      Contact( "Unit1.EmNodes".emFeedback[6].isLinked )
      Contact( "Unit1.EmNodes".emFeedback[7].isLinked )
      Coil( #StatAllEmLinked )
   END_RUNG
   // the same network as SCL:
   #StatAllEmLinked := "Unit1.EmNodes".emFeedback[0].isLinked AND "Unit1.EmNodes".emFeedback[1].isLinked AND "Unit1.EmNodes".emFeedback[2].isLinked AND "Unit1.EmNodes".emFeedback[3].isLinked AND "Unit1.EmNodes".emFeedback[4].isLinked AND "Unit1.EmNodes".emFeedback[5].isLinked AND "Unit1.EmNodes".emFeedback[6].isLinked AND "Unit1.EmNodes".emFeedback[7].isLinked;
END_REGION

REGION Network 30: Enable interfaces to control the unit
   RUNG wire#powerrail
      Move(in := #unitInterface.enableControlInterfaces, out1 => "Unit1.EmNodes".enableControlInterfaces)
   END_RUNG
   // the same network as SCL:
   "Unit1.EmNodes".enableControlInterfaces := #unitInterface.enableControlInterfaces;
END_REGION

REGION Network 31: EM Enable Check
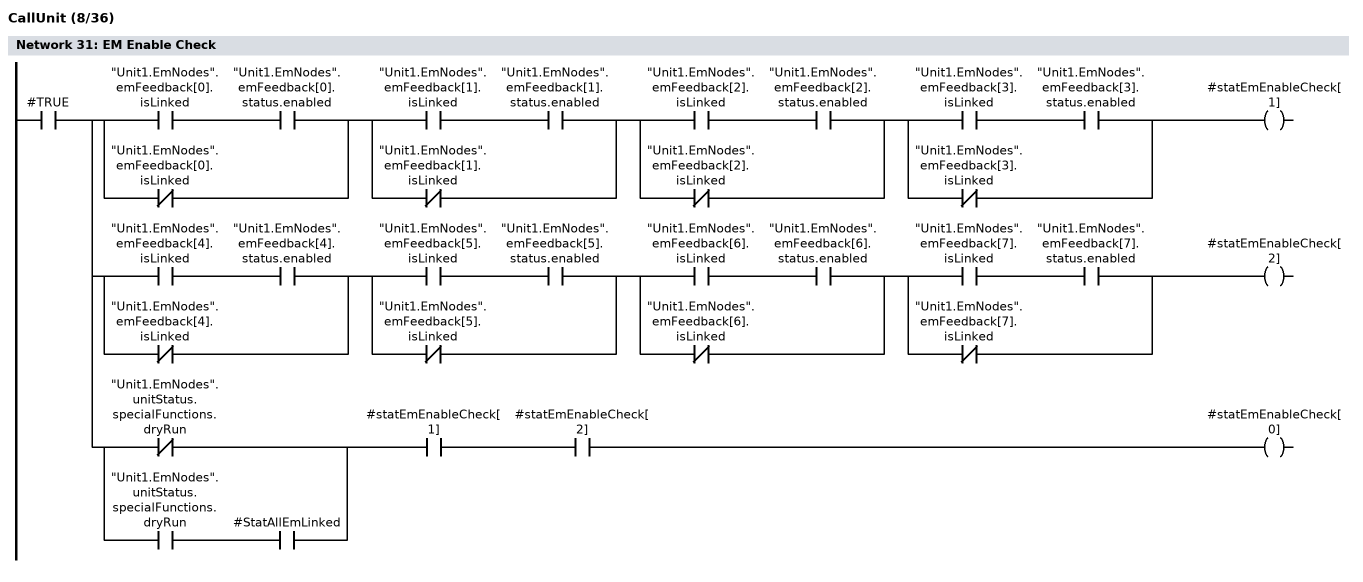
   RUNG wire#powerrail
      Contact( #TRUE )
      wire#w1
      Contact( "Unit1.EmNodes".emFeedback[0].isLinked )
      Contact( "Unit1.EmNodes".emFeedback[0].status.enabled )
      wire#w2
      Contact( "Unit1.EmNodes".emFeedback[1].isLinked )
      Contact( "Unit1.EmNodes".emFeedback[1].status.enabled )
      wire#w3
      Contact( "Unit1.EmNodes".emFeedback[2].isLinked )
      Contact( "Unit1.EmNodes".emFeedback[2].status.enabled )
      wire#w4
      Contact( "Unit1.EmNodes".emFeedback[3].isLinked )
      Contact( "Unit1.EmNodes".emFeedback[3].status.enabled )
      wire#w5
      Coil( #statEmEnableCheck[1] )
   END_RUNG
   RUNG wire#w1
      I_Contact( "Unit1.EmNodes".emFeedback[0].isLinked )
   END_RUNG wire#w2
   RUNG wire#w2
      I_Contact( "Unit1.EmNodes".emFeedback[1].isLinked )
   END_RUNG wire#w3
   RUNG wire#w3
      I_Contact( "Unit1.EmNodes".emFeedback[2].isLinked )
   END_RUNG wire#w4
   RUNG wire#w4
      I_Contact( "Unit1.EmNodes".emFeedback[3].isLinked )
   END_RUNG wire#w5
   RUNG wire#w1
      Contact( "Unit1.EmNodes".emFeedback[4].isLinked )
      Contact( "Unit1.EmNodes".emFeedback[4].status.enabled )
      wire#w6
      Contact( "Unit1.EmNodes".emFeedback[5].isLinked )
      Contact( "Unit1.EmNodes".emFeedback[5].status.enabled )
      wire#w7
      Contact( "Unit1.EmNodes".emFeedback[6].isLinked )
      Contact( "Unit1.EmNodes".emFeedback[6].status.enabled )
      wire#w8
      Contact( "Unit1.EmNodes".emFeedback[7].isLinked )
      Contact( "Unit1.EmNodes".emFeedback[7].status.enabled )
      wire#w9
      Coil( #statEmEnableCheck[2] )
   END_RUNG
   RUNG wire#w1
      I_Contact( "Unit1.EmNodes".emFeedback[4].isLinked )
   END_RUNG wire#w6
   RUNG wire#w6
      I_Contact( "Unit1.EmNodes".emFeedback[5].isLinked )
   END_RUNG wire#w7
   RUNG wire#w7
      I_Contact( "Unit1.EmNodes".emFeedback[6].isLinked )
   END_RUNG wire#w8
   RUNG wire#w8
      I_Contact( "Unit1.EmNodes".emFeedback[7].isLinked )
   END_RUNG wire#w9
   RUNG wire#w1
      I_Contact( "Unit1.EmNodes".unitStatus.specialFunctions.dryRun )
      wire#w10
      Contact( #statEmEnableCheck[1] )
      Contact( #statEmEnableCheck[2] )
      Coil( #statEmEnableCheck[0] )
   END_RUNG
   RUNG wire#w1
      Contact( "Unit1.EmNodes".unitStatus.specialFunctions.dryRun )
      Contact( #StatAllEmLinked )
   END_RUNG wire#w10
   // the same network as SCL:
   #statEmEnableCheck[1] := #TRUE AND (("Unit1.EmNodes".emFeedback[0].isLinked AND "Unit1.EmNodes".emFeedback[0].status.enabled) OR NOT "Unit1.EmNodes".emFeedback[0].isLinked) AND (("Unit1.EmNodes".emFeedback[1].isLinked AND "Unit1.EmNodes".emFeedback[1].status.enabled) OR NOT "Unit1.EmNodes".emFeedback[1].isLinked) AND (("Unit1.EmNodes".emFeedback[2].isLinked AND "Unit1.EmNodes".emFeedback[2].status.enabled) OR NOT "Unit1.EmNodes".emFeedback[2].isLinked) AND (("Unit1.EmNodes".emFeedback[3].isLinked AND "Unit1.EmNodes".emFeedback[3].status.enabled) OR NOT "Unit1.EmNodes".emFeedback[3].isLinked);
   #statEmEnableCheck[2] := #TRUE AND (("Unit1.EmNodes".emFeedback[4].isLinked AND "Unit1.EmNodes".emFeedback[4].status.enabled) OR NOT "Unit1.EmNodes".emFeedback[4].isLinked) AND (("Unit1.EmNodes".emFeedback[5].isLinked AND "Unit1.EmNodes".emFeedback[5].status.enabled) OR NOT "Unit1.EmNodes".emFeedback[5].isLinked) AND (("Unit1.EmNodes".emFeedback[6].isLinked AND "Unit1.EmNodes".emFeedback[6].status.enabled) OR NOT "Unit1.EmNodes".emFeedback[6].isLinked) AND (("Unit1.EmNodes".emFeedback[7].isLinked AND "Unit1.EmNodes".emFeedback[7].status.enabled) OR NOT "Unit1.EmNodes".emFeedback[7].isLinked);
   #statEmEnableCheck[0] := #TRUE AND (NOT "Unit1.EmNodes".unitStatus.specialFunctions.dryRun OR ("Unit1.EmNodes".unitStatus.specialFunctions.dryRun AND #StatAllEmLinked)) AND #statEmEnableCheck[1] AND #statEmEnableCheck[2];
END_REGION

REGION Network 32: Special Fuction Enable Check
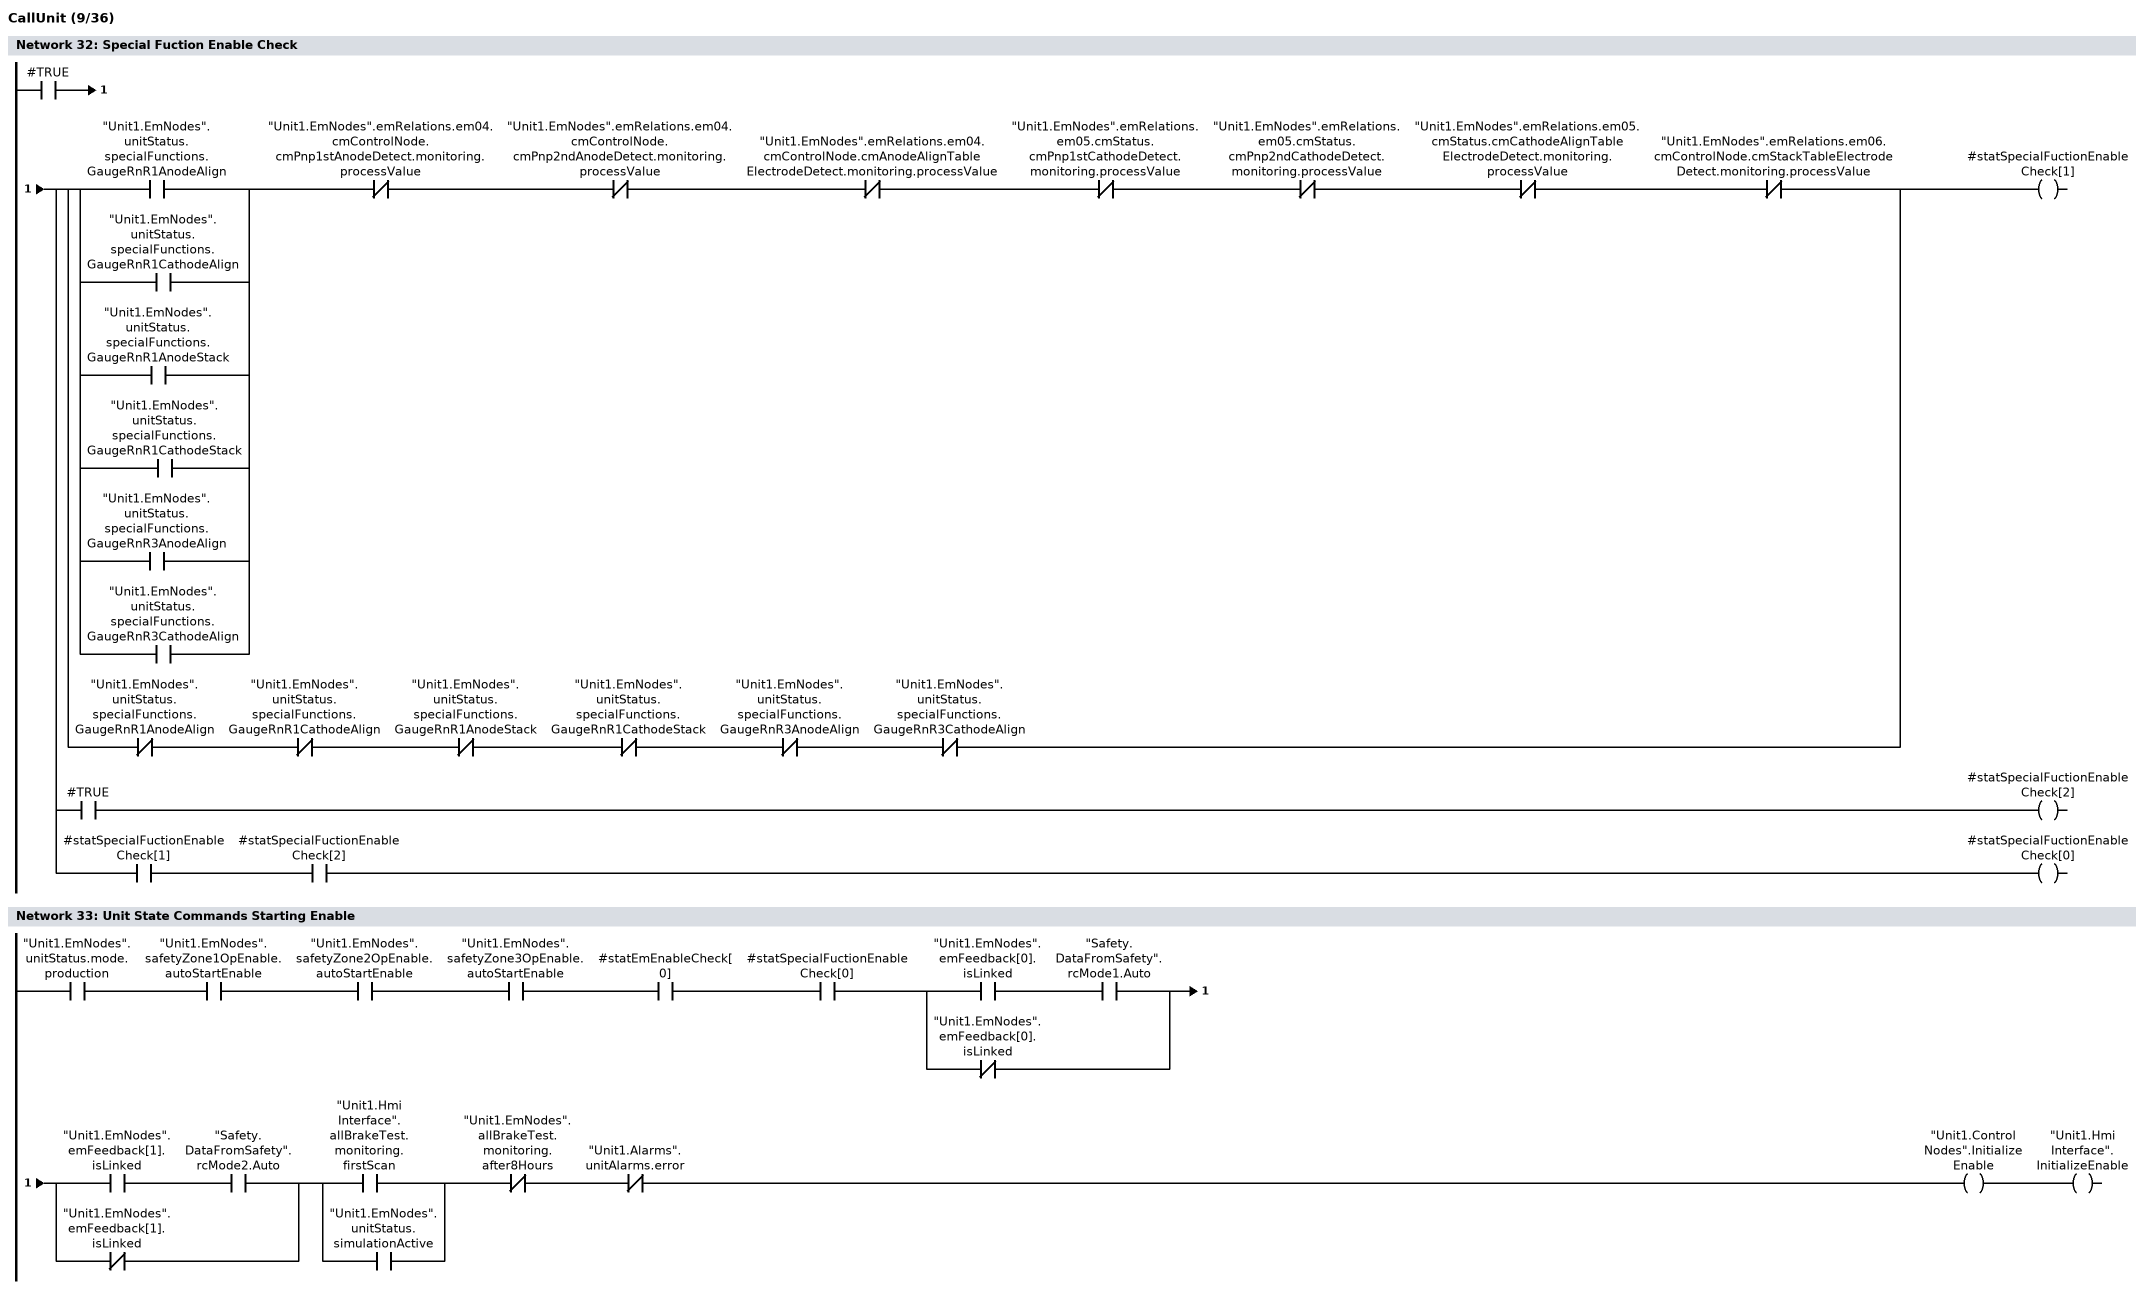
   RUNG wire#powerrail
      Contact( #TRUE )
      wire#w1
      Contact( "Unit1.EmNodes".unitStatus.specialFunctions.GaugeRnR1AnodeAlign )
      wire#w2
      I_Contact( "Unit1.EmNodes".emRelations.em04.cmControlNode.cmPnp1stAnodeDetect.monitoring.processValue )
      I_Contact( "Unit1.EmNodes".emRelations.em04.cmControlNode.cmPnp2ndAnodeDetect.monitoring.processValue )
      I_Contact( "Unit1.EmNodes".emRelations.em04.cmControlNode.cmAnodeAlignTableElectrodeDetect.monitoring.processValue )
      I_Contact( "Unit1.EmNodes".emRelations.em05.cmStatus.cmPnp1stCathodeDetect.monitoring.processValue )
      I_Contact( "Unit1.EmNodes".emRelations.em05.cmStatus.cmPnp2ndCathodeDetect.monitoring.processValue )
      I_Contact( "Unit1.EmNodes".emRelations.em05.cmStatus.cmCathodeAlignTableElectrodeDetect.monitoring.processValue )
      I_Contact( "Unit1.EmNodes".emRelations.em06.cmControlNode.cmStackTableElectrodeDetect.monitoring.processValue )
      wire#w3
      Coil( #statSpecialFuctionEnableCheck[1] )
   END_RUNG
   RUNG wire#w1
      Contact( "Unit1.EmNodes".unitStatus.specialFunctions.GaugeRnR1CathodeAlign )
   END_RUNG wire#w2
   RUNG wire#w1
      Contact( "Unit1.EmNodes".unitStatus.specialFunctions.GaugeRnR1AnodeStack )
   END_RUNG wire#w2
   RUNG wire#w1
      Contact( "Unit1.EmNodes".unitStatus.specialFunctions.GaugeRnR1CathodeStack )
   END_RUNG wire#w2
   RUNG wire#w1
      Contact( "Unit1.EmNodes".unitStatus.specialFunctions.GaugeRnR3AnodeAlign )
   END_RUNG wire#w2
   RUNG wire#w1
      Contact( "Unit1.EmNodes".unitStatus.specialFunctions.GaugeRnR3CathodeAlign )
   END_RUNG wire#w2
   RUNG wire#w1
      I_Contact( "Unit1.EmNodes".unitStatus.specialFunctions.GaugeRnR1AnodeAlign )
      I_Contact( "Unit1.EmNodes".unitStatus.specialFunctions.GaugeRnR1CathodeAlign )
      I_Contact( "Unit1.EmNodes".unitStatus.specialFunctions.GaugeRnR1AnodeStack )
      I_Contact( "Unit1.EmNodes".unitStatus.specialFunctions.GaugeRnR1CathodeStack )
      I_Contact( "Unit1.EmNodes".unitStatus.specialFunctions.GaugeRnR3AnodeAlign )
      I_Contact( "Unit1.EmNodes".unitStatus.specialFunctions.GaugeRnR3CathodeAlign )
   END_RUNG wire#w3
   RUNG wire#w1
      Contact( #TRUE )
      Coil( #statSpecialFuctionEnableCheck[2] )
   END_RUNG
   RUNG wire#w1
      Contact( #statSpecialFuctionEnableCheck[1] )
      Contact( #statSpecialFuctionEnableCheck[2] )
      Coil( #statSpecialFuctionEnableCheck[0] )
   END_RUNG
   // the same network as SCL:
   #statSpecialFuctionEnableCheck[1] := #TRUE AND ((("Unit1.EmNodes".unitStatus.specialFunctions.GaugeRnR1AnodeAlign OR "Unit1.EmNodes".unitStatus.specialFunctions.GaugeRnR1CathodeAlign OR "Unit1.EmNodes".unitStatus.specialFunctions.GaugeRnR1AnodeStack OR "Unit1.EmNodes".unitStatus.specialFunctions.GaugeRnR1CathodeStack OR "Unit1.EmNodes".unitStatus.specialFunctions.GaugeRnR3AnodeAlign OR "Unit1.EmNodes".unitStatus.specialFunctions.GaugeRnR3CathodeAlign) AND NOT "Unit1.EmNodes".emRelations.em04.cmControlNode.cmPnp1stAnodeDetect.monitoring.processValue AND NOT "Unit1.EmNodes".emRelations.em04.cmControlNode.cmPnp2ndAnodeDetect.monitoring.processValue AND NOT "Unit1.EmNodes".emRelations.em04.cmControlNode.cmAnodeAlignTableElectrodeDetect.monitoring.processValue AND NOT "Unit1.EmNodes".emRelations.em05.cmStatus.cmPnp1stCathodeDetect.monitoring.processValue AND NOT "Unit1.EmNodes".emRelations.em05.cmStatus.cmPnp2ndCathodeDetect.monitoring.processValue AND NOT "Unit1.EmNodes".emRelations.em05.cmStatus.cmCathodeAlignTableElectrodeDetect.monitoring.processValue AND NOT "Unit1.EmNodes".emRelations.em06.cmControlNode.cmStackTableElectrodeDetect.monitoring.processValue) OR (NOT "Unit1.EmNodes".unitStatus.specialFunctions.GaugeRnR1AnodeAlign AND NOT "Unit1.EmNodes".unitStatus.specialFunctions.GaugeRnR1CathodeAlign AND NOT "Unit1.EmNodes".unitStatus.specialFunctions.GaugeRnR1AnodeStack AND NOT "Unit1.EmNodes".unitStatus.specialFunctions.GaugeRnR1CathodeStack AND NOT "Unit1.EmNodes".unitStatus.specialFunctions.GaugeRnR3AnodeAlign AND NOT "Unit1.EmNodes".unitStatus.specialFunctions.GaugeRnR3CathodeAlign));
   #statSpecialFuctionEnableCheck[2] := #TRUE AND #TRUE;
   #statSpecialFuctionEnableCheck[0] := #TRUE AND #statSpecialFuctionEnableCheck[1] AND #statSpecialFuctionEnableCheck[2];
END_REGION

REGION Network 33: Unit State Commands Starting Enable
   RUNG wire#powerrail
      Contact( "Unit1.EmNodes".unitStatus.mode.production )
      Contact( "Unit1.EmNodes".safetyZone1OpEnable.autoStartEnable )
      Contact( "Unit1.EmNodes".safetyZone2OpEnable.autoStartEnable )
      Contact( "Unit1.EmNodes".safetyZone3OpEnable.autoStartEnable )
      Contact( #statEmEnableCheck[0] )
      Contact( #statSpecialFuctionEnableCheck[0] )
      wire#w1
      Contact( "Unit1.EmNodes".emFeedback[0].isLinked )
      Contact( "Safety.DataFromSafety".rcMode1.Auto )
      wire#w2
      Contact( "Unit1.EmNodes".emFeedback[1].isLinked )
      Contact( "Safety.DataFromSafety".rcMode2.Auto )
      wire#w3
      Contact( "Unit1.HmiInterface".allBrakeTest.monitoring.firstScan )
      wire#w4
      I_Contact( "Unit1.EmNodes".allBrakeTest.monitoring.after8Hours )
      I_Contact( "Unit1.Alarms".unitAlarms.error )
      Coil( "Unit1.ControlNodes".InitializeEnable )
      Coil( "Unit1.HmiInterface".InitializeEnable )
   END_RUNG
   RUNG wire#w1
      I_Contact( "Unit1.EmNodes".emFeedback[0].isLinked )
   END_RUNG wire#w2
   RUNG wire#w2
      I_Contact( "Unit1.EmNodes".emFeedback[1].isLinked )
   END_RUNG wire#w3
   RUNG wire#w3
      Contact( "Unit1.EmNodes".unitStatus.simulationActive )
   END_RUNG wire#w4
   // the same network as SCL:
   "Unit1.ControlNodes".InitializeEnable := "Unit1.EmNodes".unitStatus.mode.production AND "Unit1.EmNodes".safetyZone1OpEnable.autoStartEnable AND "Unit1.EmNodes".safetyZone2OpEnable.autoStartEnable AND "Unit1.EmNodes".safetyZone3OpEnable.autoStartEnable AND #statEmEnableCheck[0] AND #statSpecialFuctionEnableCheck[0] AND (("Unit1.EmNodes".emFeedback[0].isLinked AND "Safety.DataFromSafety".rcMode1.Auto) OR NOT "Unit1.EmNodes".emFeedback[0].isLinked) AND (("Unit1.EmNodes".emFeedback[1].isLinked AND "Safety.DataFromSafety".rcMode2.Auto) OR NOT "Unit1.EmNodes".emFeedback[1].isLinked) AND ("Unit1.HmiInterface".allBrakeTest.monitoring.firstScan OR "Unit1.EmNodes".unitStatus.simulationActive) AND NOT "Unit1.EmNodes".allBrakeTest.monitoring.after8Hours AND NOT "Unit1.Alarms".unitAlarms.error;
   "Unit1.HmiInterface".InitializeEnable := "Unit1.ControlNodes".InitializeEnable;
END_REGION

REGION Network 34: EM initialized + Homed Check
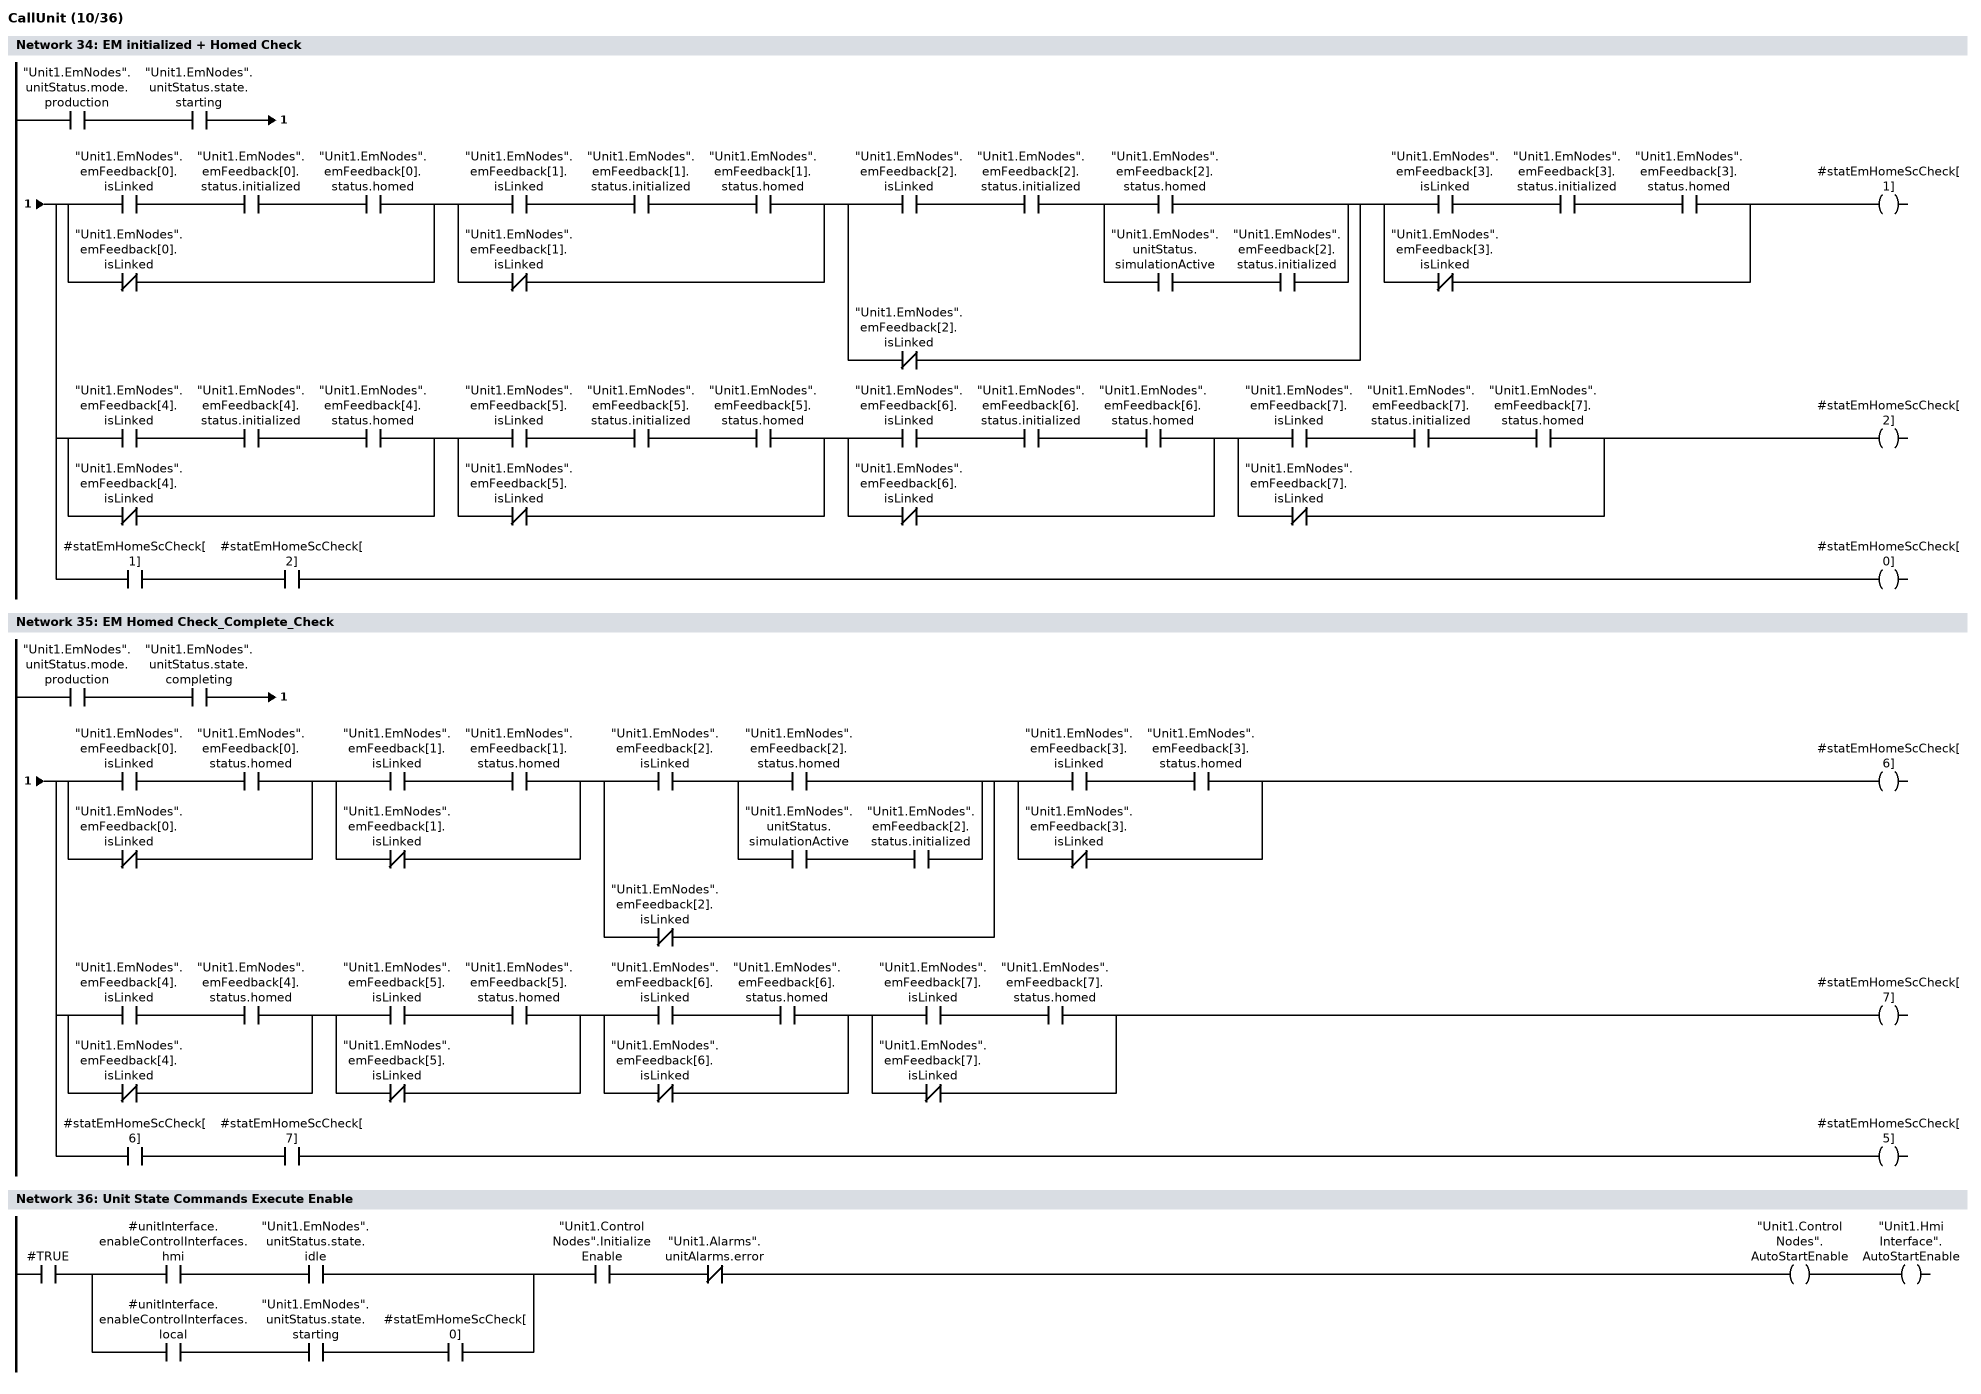
   RUNG wire#powerrail
      Contact( "Unit1.EmNodes".unitStatus.mode.production )
      Contact( "Unit1.EmNodes".unitStatus.state.starting )
      wire#w1
      Contact( "Unit1.EmNodes".emFeedback[0].isLinked )
      Contact( "Unit1.EmNodes".emFeedback[0].status.initialized )
      Contact( "Unit1.EmNodes".emFeedback[0].status.homed )
      wire#w2
      Contact( "Unit1.EmNodes".emFeedback[1].isLinked )
      Contact( "Unit1.EmNodes".emFeedback[1].status.initialized )
      Contact( "Unit1.EmNodes".emFeedback[1].status.homed )
      wire#w3
      Contact( "Unit1.EmNodes".emFeedback[2].isLinked )
      Contact( "Unit1.EmNodes".emFeedback[2].status.initialized )
      wire#w4
      Contact( "Unit1.EmNodes".emFeedback[2].status.homed )
      wire#w5
      Contact( "Unit1.EmNodes".emFeedback[3].isLinked )
      Contact( "Unit1.EmNodes".emFeedback[3].status.initialized )
      Contact( "Unit1.EmNodes".emFeedback[3].status.homed )
      wire#w6
      Coil( #statEmHomeScCheck[1] )
   END_RUNG
   RUNG wire#w1
      I_Contact( "Unit1.EmNodes".emFeedback[0].isLinked )
   END_RUNG wire#w2
   RUNG wire#w2
      I_Contact( "Unit1.EmNodes".emFeedback[1].isLinked )
   END_RUNG wire#w3
   RUNG wire#w4
      Contact( "Unit1.EmNodes".unitStatus.simulationActive )
      Contact( "Unit1.EmNodes".emFeedback[2].status.initialized )
   END_RUNG wire#w5
   RUNG wire#w3
      I_Contact( "Unit1.EmNodes".emFeedback[2].isLinked )
   END_RUNG wire#w5
   RUNG wire#w5
      I_Contact( "Unit1.EmNodes".emFeedback[3].isLinked )
   END_RUNG wire#w6
   RUNG wire#w1
      Contact( "Unit1.EmNodes".emFeedback[4].isLinked )
      Contact( "Unit1.EmNodes".emFeedback[4].status.initialized )
      Contact( "Unit1.EmNodes".emFeedback[4].status.homed )
      wire#w7
      Contact( "Unit1.EmNodes".emFeedback[5].isLinked )
      Contact( "Unit1.EmNodes".emFeedback[5].status.initialized )
      Contact( "Unit1.EmNodes".emFeedback[5].status.homed )
      wire#w8
      Contact( "Unit1.EmNodes".emFeedback[6].isLinked )
      Contact( "Unit1.EmNodes".emFeedback[6].status.initialized )
      Contact( "Unit1.EmNodes".emFeedback[6].status.homed )
      wire#w9
      Contact( "Unit1.EmNodes".emFeedback[7].isLinked )
      Contact( "Unit1.EmNodes".emFeedback[7].status.initialized )
      Contact( "Unit1.EmNodes".emFeedback[7].status.homed )
      wire#w10
      Coil( #statEmHomeScCheck[2] )
   END_RUNG
   RUNG wire#w1
      I_Contact( "Unit1.EmNodes".emFeedback[4].isLinked )
   END_RUNG wire#w7
   RUNG wire#w7
      I_Contact( "Unit1.EmNodes".emFeedback[5].isLinked )
   END_RUNG wire#w8
   RUNG wire#w8
      I_Contact( "Unit1.EmNodes".emFeedback[6].isLinked )
   END_RUNG wire#w9
   RUNG wire#w9
      I_Contact( "Unit1.EmNodes".emFeedback[7].isLinked )
   END_RUNG wire#w10
   RUNG wire#w1
      Contact( #statEmHomeScCheck[1] )
      Contact( #statEmHomeScCheck[2] )
      Coil( #statEmHomeScCheck[0] )
   END_RUNG
   // the same network as SCL:
   #_w1 := "Unit1.EmNodes".unitStatus.mode.production AND "Unit1.EmNodes".unitStatus.state.starting;
   #statEmHomeScCheck[1] := #_w1 AND (("Unit1.EmNodes".emFeedback[0].isLinked AND "Unit1.EmNodes".emFeedback[0].status.initialized AND "Unit1.EmNodes".emFeedback[0].status.homed) OR NOT "Unit1.EmNodes".emFeedback[0].isLinked) AND (("Unit1.EmNodes".emFeedback[1].isLinked AND "Unit1.EmNodes".emFeedback[1].status.initialized AND "Unit1.EmNodes".emFeedback[1].status.homed) OR NOT "Unit1.EmNodes".emFeedback[1].isLinked) AND (("Unit1.EmNodes".emFeedback[2].isLinked AND "Unit1.EmNodes".emFeedback[2].status.initialized AND ("Unit1.EmNodes".emFeedback[2].status.homed OR ("Unit1.EmNodes".unitStatus.simulationActive AND "Unit1.EmNodes".emFeedback[2].status.initialized))) OR NOT "Unit1.EmNodes".emFeedback[2].isLinked) AND (("Unit1.EmNodes".emFeedback[3].isLinked AND "Unit1.EmNodes".emFeedback[3].status.initialized AND "Unit1.EmNodes".emFeedback[3].status.homed) OR NOT "Unit1.EmNodes".emFeedback[3].isLinked);
   #statEmHomeScCheck[2] := #_w1 AND (("Unit1.EmNodes".emFeedback[4].isLinked AND "Unit1.EmNodes".emFeedback[4].status.initialized AND "Unit1.EmNodes".emFeedback[4].status.homed) OR NOT "Unit1.EmNodes".emFeedback[4].isLinked) AND (("Unit1.EmNodes".emFeedback[5].isLinked AND "Unit1.EmNodes".emFeedback[5].status.initialized AND "Unit1.EmNodes".emFeedback[5].status.homed) OR NOT "Unit1.EmNodes".emFeedback[5].isLinked) AND (("Unit1.EmNodes".emFeedback[6].isLinked AND "Unit1.EmNodes".emFeedback[6].status.initialized AND "Unit1.EmNodes".emFeedback[6].status.homed) OR NOT "Unit1.EmNodes".emFeedback[6].isLinked) AND (("Unit1.EmNodes".emFeedback[7].isLinked AND "Unit1.EmNodes".emFeedback[7].status.initialized AND "Unit1.EmNodes".emFeedback[7].status.homed) OR NOT "Unit1.EmNodes".emFeedback[7].isLinked);
   #statEmHomeScCheck[0] := #_w1 AND #statEmHomeScCheck[1] AND #statEmHomeScCheck[2];
END_REGION

REGION Network 35: EM Homed Check_Complete_Check
   RUNG wire#powerrail
      Contact( "Unit1.EmNodes".unitStatus.mode.production )
      Contact( "Unit1.EmNodes".unitStatus.state.completing )
      wire#w1
      Contact( "Unit1.EmNodes".emFeedback[0].isLinked )
      Contact( "Unit1.EmNodes".emFeedback[0].status.homed )
      wire#w2
      Contact( "Unit1.EmNodes".emFeedback[1].isLinked )
      Contact( "Unit1.EmNodes".emFeedback[1].status.homed )
      wire#w3
      Contact( "Unit1.EmNodes".emFeedback[2].isLinked )
      wire#w4
      Contact( "Unit1.EmNodes".emFeedback[2].status.homed )
      wire#w5
      Contact( "Unit1.EmNodes".emFeedback[3].isLinked )
      Contact( "Unit1.EmNodes".emFeedback[3].status.homed )
      wire#w6
      Coil( #statEmHomeScCheck[6] )
   END_RUNG
   RUNG wire#w1
      I_Contact( "Unit1.EmNodes".emFeedback[0].isLinked )
   END_RUNG wire#w2
   RUNG wire#w2
      I_Contact( "Unit1.EmNodes".emFeedback[1].isLinked )
   END_RUNG wire#w3
   RUNG wire#w4
      Contact( "Unit1.EmNodes".unitStatus.simulationActive )
      Contact( "Unit1.EmNodes".emFeedback[2].status.initialized )
   END_RUNG wire#w5
   RUNG wire#w3
      I_Contact( "Unit1.EmNodes".emFeedback[2].isLinked )
   END_RUNG wire#w5
   RUNG wire#w5
      I_Contact( "Unit1.EmNodes".emFeedback[3].isLinked )
   END_RUNG wire#w6
   RUNG wire#w1
      Contact( "Unit1.EmNodes".emFeedback[4].isLinked )
      Contact( "Unit1.EmNodes".emFeedback[4].status.homed )
      wire#w7
      Contact( "Unit1.EmNodes".emFeedback[5].isLinked )
      Contact( "Unit1.EmNodes".emFeedback[5].status.homed )
      wire#w8
      Contact( "Unit1.EmNodes".emFeedback[6].isLinked )
      Contact( "Unit1.EmNodes".emFeedback[6].status.homed )
      wire#w9
      Contact( "Unit1.EmNodes".emFeedback[7].isLinked )
      Contact( "Unit1.EmNodes".emFeedback[7].status.homed )
      wire#w10
      Coil( #statEmHomeScCheck[7] )
   END_RUNG
   RUNG wire#w1
      I_Contact( "Unit1.EmNodes".emFeedback[4].isLinked )
   END_RUNG wire#w7
   RUNG wire#w7
      I_Contact( "Unit1.EmNodes".emFeedback[5].isLinked )
   END_RUNG wire#w8
   RUNG wire#w8
      I_Contact( "Unit1.EmNodes".emFeedback[6].isLinked )
   END_RUNG wire#w9
   RUNG wire#w9
      I_Contact( "Unit1.EmNodes".emFeedback[7].isLinked )
   END_RUNG wire#w10
   RUNG wire#w1
      Contact( #statEmHomeScCheck[6] )
      Contact( #statEmHomeScCheck[7] )
      Coil( #statEmHomeScCheck[5] )
   END_RUNG
   // the same network as SCL:
   #_w1 := "Unit1.EmNodes".unitStatus.mode.production AND "Unit1.EmNodes".unitStatus.state.completing;
   #statEmHomeScCheck[6] := #_w1 AND (("Unit1.EmNodes".emFeedback[0].isLinked AND "Unit1.EmNodes".emFeedback[0].status.homed) OR NOT "Unit1.EmNodes".emFeedback[0].isLinked) AND (("Unit1.EmNodes".emFeedback[1].isLinked AND "Unit1.EmNodes".emFeedback[1].status.homed) OR NOT "Unit1.EmNodes".emFeedback[1].isLinked) AND (("Unit1.EmNodes".emFeedback[2].isLinked AND ("Unit1.EmNodes".emFeedback[2].status.homed OR ("Unit1.EmNodes".unitStatus.simulationActive AND "Unit1.EmNodes".emFeedback[2].status.initialized))) OR NOT "Unit1.EmNodes".emFeedback[2].isLinked) AND (("Unit1.EmNodes".emFeedback[3].isLinked AND "Unit1.EmNodes".emFeedback[3].status.homed) OR NOT "Unit1.EmNodes".emFeedback[3].isLinked);
   #statEmHomeScCheck[7] := #_w1 AND (("Unit1.EmNodes".emFeedback[4].isLinked AND "Unit1.EmNodes".emFeedback[4].status.homed) OR NOT "Unit1.EmNodes".emFeedback[4].isLinked) AND (("Unit1.EmNodes".emFeedback[5].isLinked AND "Unit1.EmNodes".emFeedback[5].status.homed) OR NOT "Unit1.EmNodes".emFeedback[5].isLinked) AND (("Unit1.EmNodes".emFeedback[6].isLinked AND "Unit1.EmNodes".emFeedback[6].status.homed) OR NOT "Unit1.EmNodes".emFeedback[6].isLinked) AND (("Unit1.EmNodes".emFeedback[7].isLinked AND "Unit1.EmNodes".emFeedback[7].status.homed) OR NOT "Unit1.EmNodes".emFeedback[7].isLinked);
   #statEmHomeScCheck[5] := #_w1 AND #statEmHomeScCheck[6] AND #statEmHomeScCheck[7];
END_REGION

REGION Network 36: Unit State Commands Execute Enable
   RUNG wire#powerrail
      Contact( #TRUE )
      wire#w1
      Contact( #unitInterface.enableControlInterfaces.hmi )
      Contact( "Unit1.EmNodes".unitStatus.state.idle )
      wire#w2
      Contact( "Unit1.ControlNodes".InitializeEnable )
      I_Contact( "Unit1.Alarms".unitAlarms.error )
      Coil( "Unit1.ControlNodes".AutoStartEnable )
      Coil( "Unit1.HmiInterface".AutoStartEnable )
   END_RUNG
   RUNG wire#w1
      Contact( #unitInterface.enableControlInterfaces.local )
      Contact( "Unit1.EmNodes".unitStatus.state.starting )
      Contact( #statEmHomeScCheck[0] )
   END_RUNG wire#w2
   // the same network as SCL:
   "Unit1.ControlNodes".AutoStartEnable := #TRUE AND ((#unitInterface.enableControlInterfaces.hmi AND "Unit1.EmNodes".unitStatus.state.idle) OR (#unitInterface.enableControlInterfaces.local AND "Unit1.EmNodes".unitStatus.state.starting AND #statEmHomeScCheck[0])) AND "Unit1.ControlNodes".InitializeEnable AND NOT "Unit1.Alarms".unitAlarms.error;
   "Unit1.HmiInterface".AutoStartEnable := "Unit1.ControlNodes".AutoStartEnable;
END_REGION

REGION Network 37: Stacklight Lamp
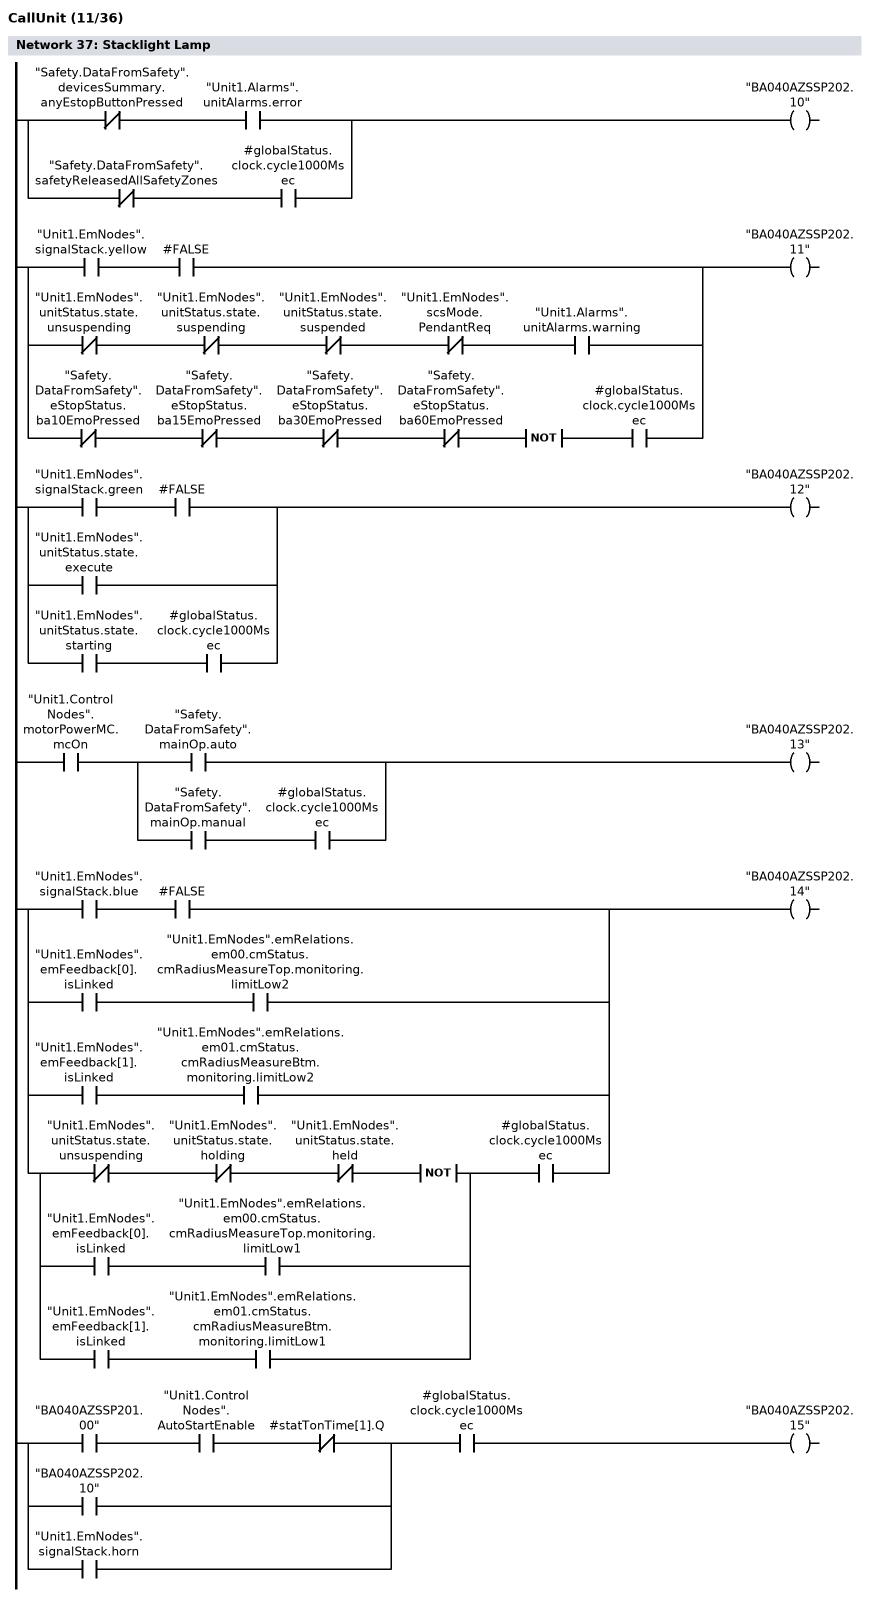
   RUNG wire#powerrail
      I_Contact( "Safety.DataFromSafety".devicesSummary.anyEstopButtonPressed )
      Contact( "Unit1.Alarms".unitAlarms.error )
      wire#w1
      Coil( "BA040AZSSP202.10" )
   END_RUNG
   RUNG wire#powerrail
      I_Contact( "Safety.DataFromSafety".safetyReleasedAllSafetyZones )
      Contact( #globalStatus.clock.cycle1000Msec )
   END_RUNG wire#w1
   RUNG wire#powerrail
      Contact( "Unit1.EmNodes".signalStack.yellow )
      Contact( #FALSE )
      wire#w2
      Coil( "BA040AZSSP202.11" )
   END_RUNG
   RUNG wire#powerrail
      I_Contact( "Unit1.EmNodes".unitStatus.state.unsuspending )
      I_Contact( "Unit1.EmNodes".unitStatus.state.suspending )
      I_Contact( "Unit1.EmNodes".unitStatus.state.suspended )
      I_Contact( "Unit1.EmNodes".scsMode.PendantReq )
      Contact( "Unit1.Alarms".unitAlarms.warning )
   END_RUNG wire#w2
   RUNG wire#powerrail
      I_Contact( "Safety.DataFromSafety".eStopStatus.ba10EmoPressed )
      I_Contact( "Safety.DataFromSafety".eStopStatus.ba15EmoPressed )
      I_Contact( "Safety.DataFromSafety".eStopStatus.ba30EmoPressed )
      I_Contact( "Safety.DataFromSafety".eStopStatus.ba60EmoPressed )
      Not()
      Contact( #globalStatus.clock.cycle1000Msec )
   END_RUNG wire#w2
   RUNG wire#powerrail
      Contact( "Unit1.EmNodes".signalStack.green )
      Contact( #FALSE )
      wire#w3
      Coil( "BA040AZSSP202.12" )
   END_RUNG
   RUNG wire#powerrail
      Contact( "Unit1.EmNodes".unitStatus.state.execute )
   END_RUNG wire#w3
   RUNG wire#powerrail
      Contact( "Unit1.EmNodes".unitStatus.state.starting )
      Contact( #globalStatus.clock.cycle1000Msec )
   END_RUNG wire#w3
   RUNG wire#powerrail
      Contact( "Unit1.ControlNodes".motorPowerMC.mcOn )
      wire#w4
      Contact( "Safety.DataFromSafety".mainOp.auto )
      wire#w5
      Coil( "BA040AZSSP202.13" )
   END_RUNG
   RUNG wire#w4
      Contact( "Safety.DataFromSafety".mainOp.manual )
      Contact( #globalStatus.clock.cycle1000Msec )
   END_RUNG wire#w5
   RUNG wire#powerrail
      Contact( "Unit1.EmNodes".signalStack.blue )
      Contact( #FALSE )
      wire#w6
      Coil( "BA040AZSSP202.14" )
   END_RUNG
   RUNG wire#powerrail
      Contact( "Unit1.EmNodes".emFeedback[0].isLinked )
      Contact( "Unit1.EmNodes".emRelations.em00.cmStatus.cmRadiusMeasureTop.monitoring.limitLow2 )
   END_RUNG wire#w6
   RUNG wire#powerrail
      Contact( "Unit1.EmNodes".emFeedback[1].isLinked )
      Contact( "Unit1.EmNodes".emRelations.em01.cmStatus.cmRadiusMeasureBtm.monitoring.limitLow2 )
   END_RUNG wire#w6
   RUNG wire#powerrail
      I_Contact( "Unit1.EmNodes".unitStatus.state.unsuspending )
      I_Contact( "Unit1.EmNodes".unitStatus.state.holding )
      I_Contact( "Unit1.EmNodes".unitStatus.state.held )
      Not()
      wire#w7
      Contact( #globalStatus.clock.cycle1000Msec )
   END_RUNG wire#w6
   RUNG wire#powerrail
      Contact( "Unit1.EmNodes".emFeedback[0].isLinked )
      Contact( "Unit1.EmNodes".emRelations.em00.cmStatus.cmRadiusMeasureTop.monitoring.limitLow1 )
   END_RUNG wire#w7
   RUNG wire#powerrail
      Contact( "Unit1.EmNodes".emFeedback[1].isLinked )
      Contact( "Unit1.EmNodes".emRelations.em01.cmStatus.cmRadiusMeasureBtm.monitoring.limitLow1 )
   END_RUNG wire#w7
   RUNG wire#powerrail
      Contact( "BA040AZSSP201.00" )
      Contact( "Unit1.ControlNodes".AutoStartEnable )
      I_Contact( #statTonTime[1].Q )
      wire#w8
      Contact( #globalStatus.clock.cycle1000Msec )
      Coil( "BA040AZSSP202.15" )
   END_RUNG
   RUNG wire#powerrail
      Contact( "BA040AZSSP202.10" )
   END_RUNG wire#w8
   RUNG wire#powerrail
      Contact( "Unit1.EmNodes".signalStack.horn )
   END_RUNG wire#w8
   // the same network as SCL:
   "BA040AZSSP202.10" := (NOT "Safety.DataFromSafety".devicesSummary.anyEstopButtonPressed AND "Unit1.Alarms".unitAlarms.error) OR (NOT "Safety.DataFromSafety".safetyReleasedAllSafetyZones AND #globalStatus.clock.cycle1000Msec);
   "BA040AZSSP202.11" := ("Unit1.EmNodes".signalStack.yellow AND #FALSE) OR (NOT "Unit1.EmNodes".unitStatus.state.unsuspending AND NOT "Unit1.EmNodes".unitStatus.state.suspending AND NOT "Unit1.EmNodes".unitStatus.state.suspended AND NOT "Unit1.EmNodes".scsMode.PendantReq AND "Unit1.Alarms".unitAlarms.warning) OR (NOT (NOT "Safety.DataFromSafety".eStopStatus.ba10EmoPressed AND NOT "Safety.DataFromSafety".eStopStatus.ba15EmoPressed AND NOT "Safety.DataFromSafety".eStopStatus.ba30EmoPressed AND NOT "Safety.DataFromSafety".eStopStatus.ba60EmoPressed) AND #globalStatus.clock.cycle1000Msec);
   "BA040AZSSP202.12" := ("Unit1.EmNodes".signalStack.green AND #FALSE) OR "Unit1.EmNodes".unitStatus.state.execute OR ("Unit1.EmNodes".unitStatus.state.starting AND #globalStatus.clock.cycle1000Msec);
   "BA040AZSSP202.13" := "Unit1.ControlNodes".motorPowerMC.mcOn AND ("Safety.DataFromSafety".mainOp.auto OR ("Safety.DataFromSafety".mainOp.manual AND #globalStatus.clock.cycle1000Msec));
   "BA040AZSSP202.14" := ("Unit1.EmNodes".signalStack.blue AND #FALSE) OR ("Unit1.EmNodes".emFeedback[0].isLinked AND "Unit1.EmNodes".emRelations.em00.cmStatus.cmRadiusMeasureTop.monitoring.limitLow2) OR ("Unit1.EmNodes".emFeedback[1].isLinked AND "Unit1.EmNodes".emRelations.em01.cmStatus.cmRadiusMeasureBtm.monitoring.limitLow2) OR ((NOT (NOT "Unit1.EmNodes".unitStatus.state.unsuspending AND NOT "Unit1.EmNodes".unitStatus.state.holding AND NOT "Unit1.EmNodes".unitStatus.state.held) OR ("Unit1.EmNodes".emFeedback[0].isLinked AND "Unit1.EmNodes".emRelations.em00.cmStatus.cmRadiusMeasureTop.monitoring.limitLow1) OR ("Unit1.EmNodes".emFeedback[1].isLinked AND "Unit1.EmNodes".emRelations.em01.cmStatus.cmRadiusMeasureBtm.monitoring.limitLow1)) AND #globalStatus.clock.cycle1000Msec);
   "BA040AZSSP202.15" := (("BA040AZSSP201.00" AND "Unit1.ControlNodes".AutoStartEnable AND NOT #statTonTime[1].Q) OR "BA040AZSSP202.10" OR "Unit1.EmNodes".signalStack.horn) AND #globalStatus.clock.cycle1000Msec;
END_REGION

REGION Network 38: Main Op Local Control
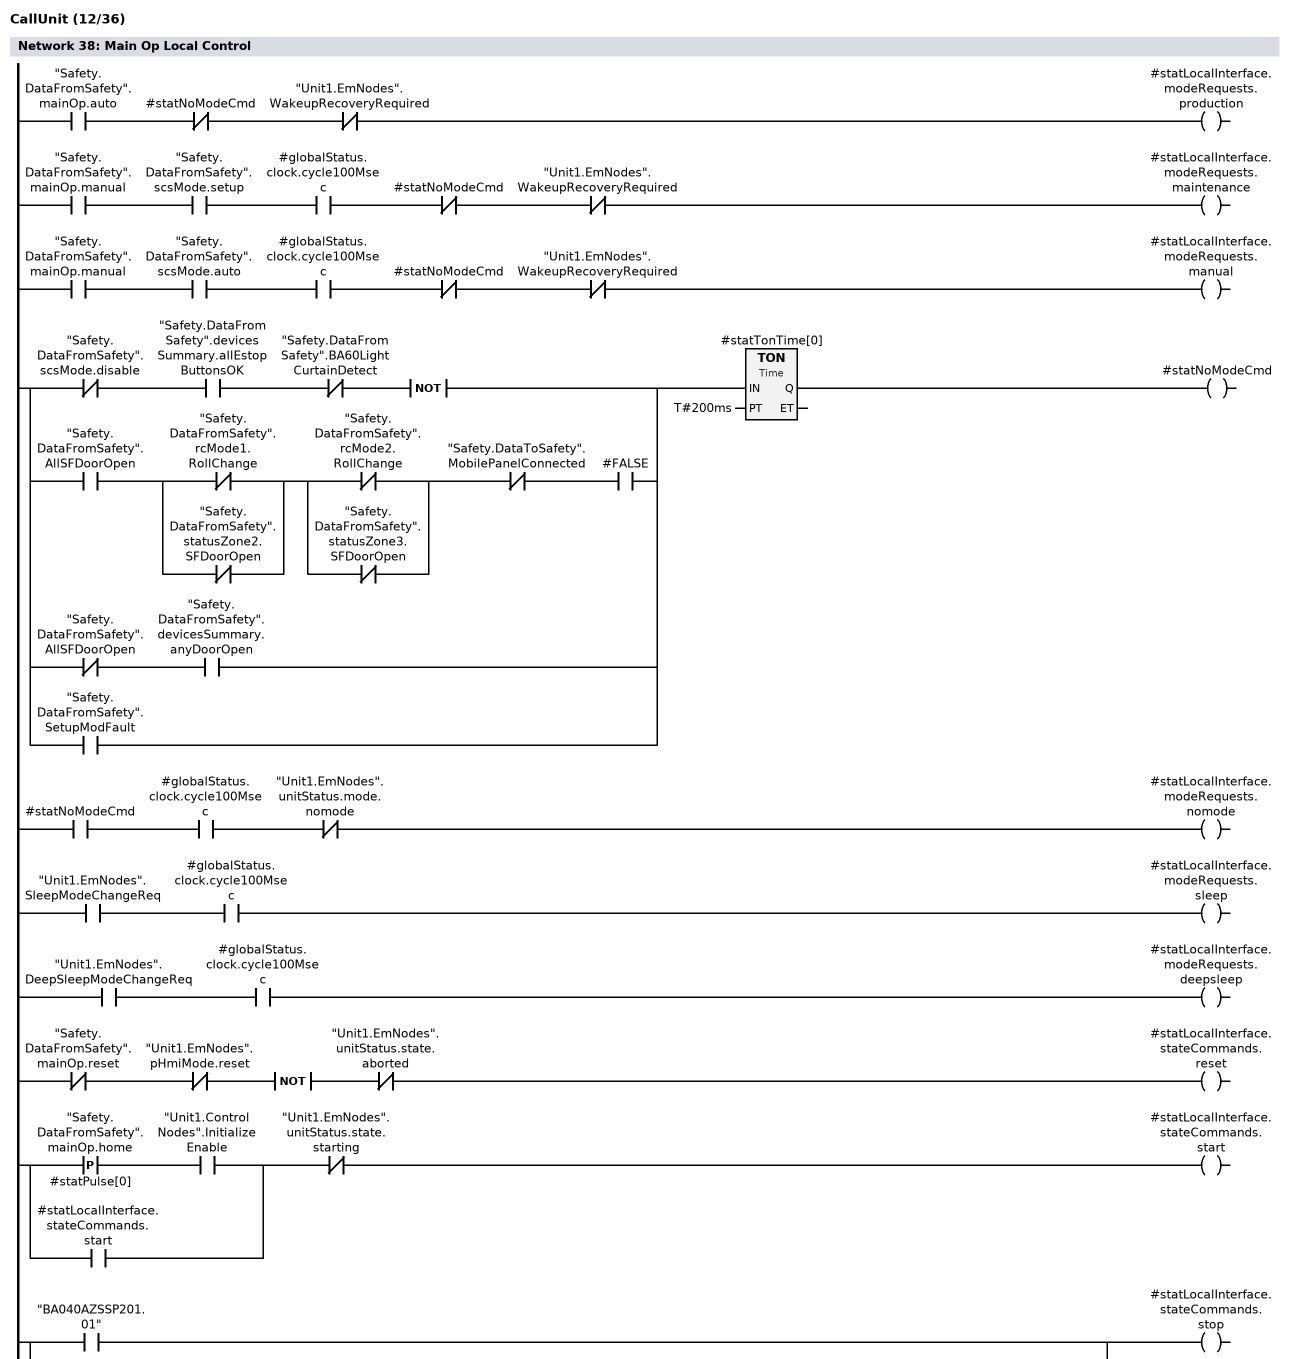
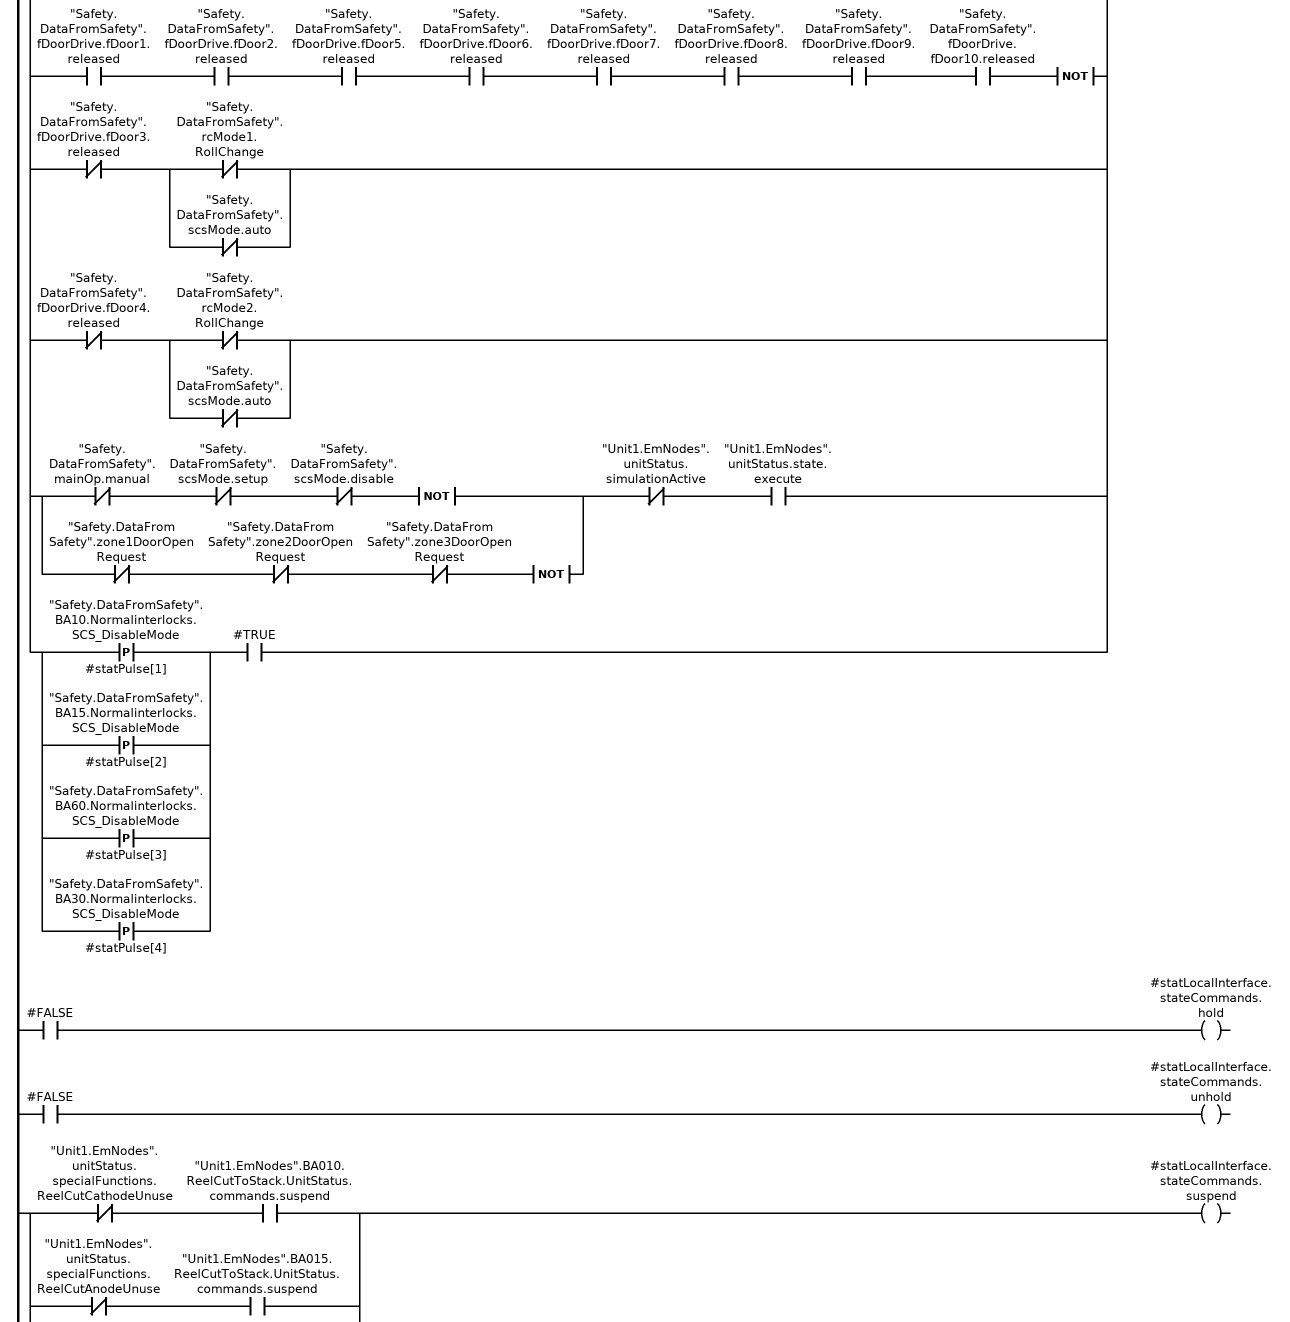
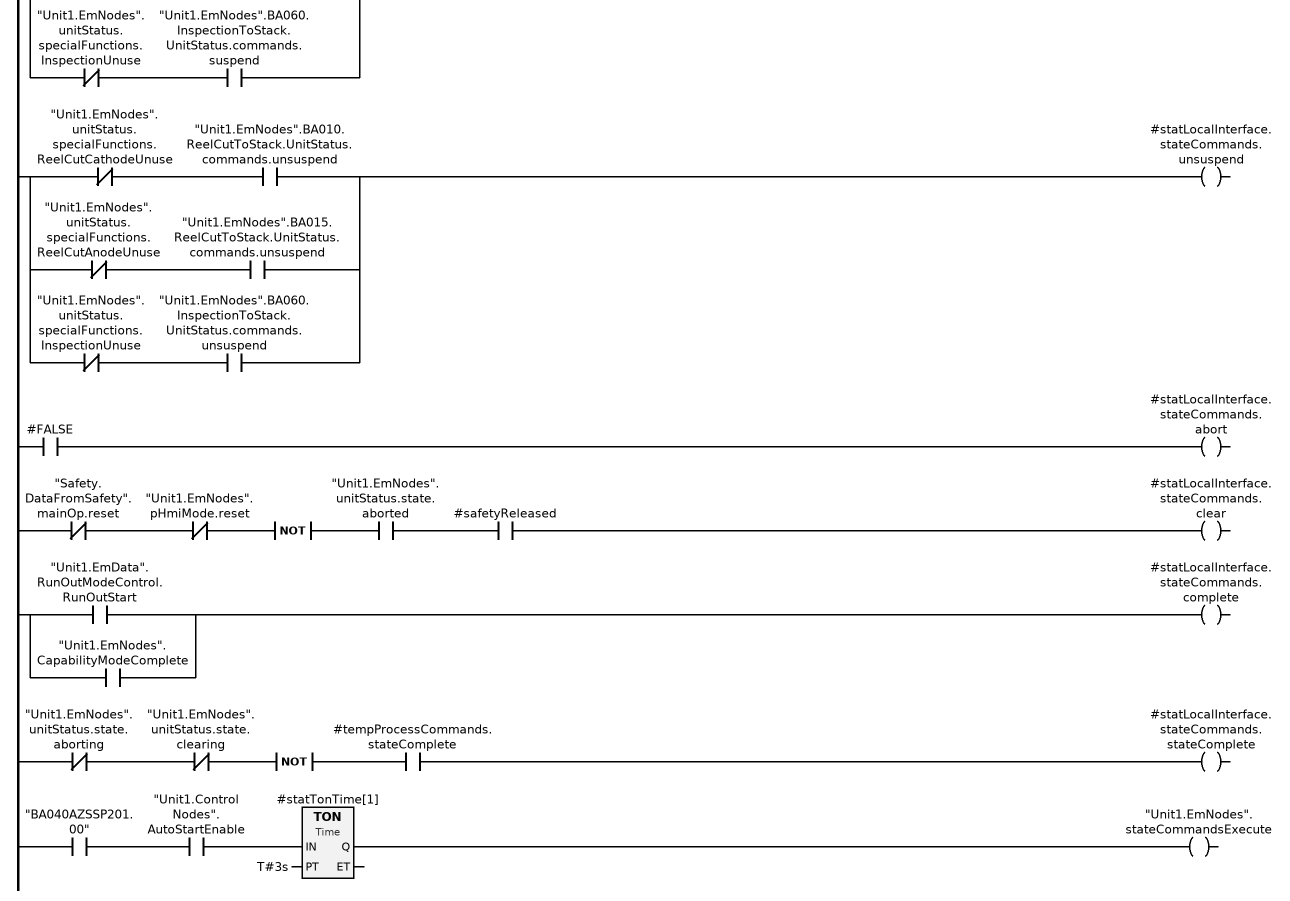
   RUNG wire#powerrail
      Contact( "Safety.DataFromSafety".mainOp.auto )
      I_Contact( #statNoModeCmd )
      I_Contact( "Unit1.EmNodes".WakeupRecoveryRequired )
      Coil( #statLocalInterface.modeRequests.production )
   END_RUNG
   RUNG wire#powerrail
      Contact( "Safety.DataFromSafety".mainOp.manual )
      Contact( "Safety.DataFromSafety".scsMode.setup )
      Contact( #globalStatus.clock.cycle100Msec )
      I_Contact( #statNoModeCmd )
      I_Contact( "Unit1.EmNodes".WakeupRecoveryRequired )
      Coil( #statLocalInterface.modeRequests.maintenance )
   END_RUNG
   RUNG wire#powerrail
      Contact( "Safety.DataFromSafety".mainOp.manual )
      Contact( "Safety.DataFromSafety".scsMode.auto )
      Contact( #globalStatus.clock.cycle100Msec )
      I_Contact( #statNoModeCmd )
      I_Contact( "Unit1.EmNodes".WakeupRecoveryRequired )
      Coil( #statLocalInterface.modeRequests.manual )
   END_RUNG
   RUNG wire#powerrail
      I_Contact( "Safety.DataFromSafety".scsMode.disable )
      Contact( "Safety.DataFromSafety".devicesSummary.allEstopButtonsOK )
      I_Contact( "Safety.DataFromSafety".BA60LightCurtainDetect )
      Not()
      wire#w1
      { S7_Templates := "time_type := Time" } #statTonTime[0].TON(pt := T#200ms, et =>)
      Coil( #statNoModeCmd )
   END_RUNG
   RUNG wire#powerrail
      Contact( "Safety.DataFromSafety".AllSFDoorOpen )
      wire#w2
      I_Contact( "Safety.DataFromSafety".rcMode1.RollChange )
      wire#w3
      I_Contact( "Safety.DataFromSafety".rcMode2.RollChange )
      wire#w4
      I_Contact( "Safety.DataToSafety".MobilePanelConnected )
      Contact( #FALSE )
   END_RUNG wire#w1
   RUNG wire#w2
      I_Contact( "Safety.DataFromSafety".statusZone2.SFDoorOpen )
   END_RUNG wire#w3
   RUNG wire#w3
      I_Contact( "Safety.DataFromSafety".statusZone3.SFDoorOpen )
   END_RUNG wire#w4
   RUNG wire#powerrail
      I_Contact( "Safety.DataFromSafety".AllSFDoorOpen )
      Contact( "Safety.DataFromSafety".devicesSummary.anyDoorOpen )
   END_RUNG wire#w1
   RUNG wire#powerrail
      Contact( "Safety.DataFromSafety".SetupModFault )
   END_RUNG wire#w1
   RUNG wire#powerrail
      Contact( #statNoModeCmd )
      Contact( #globalStatus.clock.cycle100Msec )
      I_Contact( "Unit1.EmNodes".unitStatus.mode.nomode )
      Coil( #statLocalInterface.modeRequests.nomode )
   END_RUNG
   RUNG wire#powerrail
      Contact( "Unit1.EmNodes".SleepModeChangeReq )
      Contact( #globalStatus.clock.cycle100Msec )
      Coil( #statLocalInterface.modeRequests.sleep )
   END_RUNG
   RUNG wire#powerrail
      Contact( "Unit1.EmNodes".DeepSleepModeChangeReq )
      Contact( #globalStatus.clock.cycle100Msec )
      Coil( #statLocalInterface.modeRequests.deepsleep )
   END_RUNG
   RUNG wire#powerrail
      I_Contact( "Safety.DataFromSafety".mainOp.reset )
      I_Contact( "Unit1.EmNodes".pHmiMode.reset )
      Not()
      I_Contact( "Unit1.EmNodes".unitStatus.state.aborted )
      Coil( #statLocalInterface.stateCommands.reset )
   END_RUNG
   RUNG wire#powerrail
      P_Contact(operand := "Safety.DataFromSafety".mainOp.home, bit := #statPulse[0])
      Contact( "Unit1.ControlNodes".InitializeEnable )
      wire#w5
      I_Contact( "Unit1.EmNodes".unitStatus.state.starting )
      Coil( #statLocalInterface.stateCommands.start )
   END_RUNG
   RUNG wire#powerrail
      Contact( #statLocalInterface.stateCommands.start )
   END_RUNG wire#w5
   RUNG wire#powerrail
      Contact( "BA040AZSSP201.01" )
      wire#w6
      Coil( #statLocalInterface.stateCommands.stop )
   END_RUNG
   RUNG wire#powerrail
      Contact( "Safety.DataFromSafety".fDoorDrive.fDoor1.released )
      Contact( "Safety.DataFromSafety".fDoorDrive.fDoor2.released )
      Contact( "Safety.DataFromSafety".fDoorDrive.fDoor5.released )
      Contact( "Safety.DataFromSafety".fDoorDrive.fDoor6.released )
      Contact( "Safety.DataFromSafety".fDoorDrive.fDoor7.released )
      Contact( "Safety.DataFromSafety".fDoorDrive.fDoor8.released )
      Contact( "Safety.DataFromSafety".fDoorDrive.fDoor9.released )
      Contact( "Safety.DataFromSafety".fDoorDrive.fDoor10.released )
      Not()
   END_RUNG wire#w6
   RUNG wire#powerrail
      I_Contact( "Safety.DataFromSafety".fDoorDrive.fDoor3.released )
      wire#w7
      I_Contact( "Safety.DataFromSafety".rcMode1.RollChange )
   END_RUNG wire#w6
   RUNG wire#w7
      I_Contact( "Safety.DataFromSafety".scsMode.auto )
   END_RUNG wire#w6
   RUNG wire#powerrail
      I_Contact( "Safety.DataFromSafety".fDoorDrive.fDoor4.released )
      wire#w8
      I_Contact( "Safety.DataFromSafety".rcMode2.RollChange )
   END_RUNG wire#w6
   RUNG wire#w8
      I_Contact( "Safety.DataFromSafety".scsMode.auto )
   END_RUNG wire#w6
   RUNG wire#powerrail
      I_Contact( "Safety.DataFromSafety".mainOp.manual )
      I_Contact( "Safety.DataFromSafety".scsMode.setup )
      I_Contact( "Safety.DataFromSafety".scsMode.disable )
      Not()
      wire#w9
      I_Contact( "Unit1.EmNodes".unitStatus.simulationActive )
      Contact( "Unit1.EmNodes".unitStatus.state.execute )
   END_RUNG wire#w6
   RUNG wire#powerrail
      I_Contact( "Safety.DataFromSafety".zone1DoorOpenRequest )
      I_Contact( "Safety.DataFromSafety".zone2DoorOpenRequest )
      I_Contact( "Safety.DataFromSafety".zone3DoorOpenRequest )
      Not()
   END_RUNG wire#w9
   RUNG wire#powerrail
      P_Contact(operand := "Safety.DataFromSafety".BA10.Normalinterlocks.SCS_DisableMode, bit := #statPulse[1])
      wire#w10
      Contact( #TRUE )
   END_RUNG wire#w6
   RUNG wire#powerrail
      P_Contact(operand := "Safety.DataFromSafety".BA15.Normalinterlocks.SCS_DisableMode, bit := #statPulse[2])
   END_RUNG wire#w10
   RUNG wire#powerrail
      P_Contact(operand := "Safety.DataFromSafety".BA60.Normalinterlocks.SCS_DisableMode, bit := #statPulse[3])
   END_RUNG wire#w10
   RUNG wire#powerrail
      P_Contact(operand := "Safety.DataFromSafety".BA30.Normalinterlocks.SCS_DisableMode, bit := #statPulse[4])
   END_RUNG wire#w10
   RUNG wire#powerrail
      Contact( #FALSE )
      Coil( #statLocalInterface.stateCommands.hold )
   END_RUNG
   RUNG wire#powerrail
      Contact( #FALSE )
      Coil( #statLocalInterface.stateCommands.unhold )
   END_RUNG
   RUNG wire#powerrail
      I_Contact( "Unit1.EmNodes".unitStatus.specialFunctions.ReelCutCathodeUnuse )
      Contact( "Unit1.EmNodes".BA010.ReelCutToStack.UnitStatus.commands.suspend )
      wire#w11
      Coil( #statLocalInterface.stateCommands.suspend )
   END_RUNG
   RUNG wire#powerrail
      I_Contact( "Unit1.EmNodes".unitStatus.specialFunctions.ReelCutAnodeUnuse )
      Contact( "Unit1.EmNodes".BA015.ReelCutToStack.UnitStatus.commands.suspend )
   END_RUNG wire#w11
   RUNG wire#powerrail
      I_Contact( "Unit1.EmNodes".unitStatus.specialFunctions.InspectionUnuse )
      Contact( "Unit1.EmNodes".BA060.InspectionToStack.UnitStatus.commands.suspend )
   END_RUNG wire#w11
   RUNG wire#powerrail
      I_Contact( "Unit1.EmNodes".unitStatus.specialFunctions.ReelCutCathodeUnuse )
      Contact( "Unit1.EmNodes".BA010.ReelCutToStack.UnitStatus.commands.unsuspend )
      wire#w12
      Coil( #statLocalInterface.stateCommands.unsuspend )
   END_RUNG
   RUNG wire#powerrail
      I_Contact( "Unit1.EmNodes".unitStatus.specialFunctions.ReelCutAnodeUnuse )
      Contact( "Unit1.EmNodes".BA015.ReelCutToStack.UnitStatus.commands.unsuspend )
   END_RUNG wire#w12
   RUNG wire#powerrail
      I_Contact( "Unit1.EmNodes".unitStatus.specialFunctions.InspectionUnuse )
      Contact( "Unit1.EmNodes".BA060.InspectionToStack.UnitStatus.commands.unsuspend )
   END_RUNG wire#w12
   RUNG wire#powerrail
      Contact( #FALSE )
      Coil( #statLocalInterface.stateCommands.abort )
   END_RUNG
   RUNG wire#powerrail
      I_Contact( "Safety.DataFromSafety".mainOp.reset )
      I_Contact( "Unit1.EmNodes".pHmiMode.reset )
      Not()
      Contact( "Unit1.EmNodes".unitStatus.state.aborted )
      Contact( #safetyReleased )
      Coil( #statLocalInterface.stateCommands.clear )
   END_RUNG
   RUNG wire#powerrail
      Contact( "Unit1.EmData".RunOutModeControl.RunOutStart )
      wire#w13
      Coil( #statLocalInterface.stateCommands.complete )
   END_RUNG
   RUNG wire#powerrail
      Contact( "Unit1.EmNodes".CapabilityModeComplete )
   END_RUNG wire#w13
   RUNG wire#powerrail
      I_Contact( "Unit1.EmNodes".unitStatus.state.aborting )
      I_Contact( "Unit1.EmNodes".unitStatus.state.clearing )
      Not()
      Contact( #tempProcessCommands.stateComplete )
      Coil( #statLocalInterface.stateCommands.stateComplete )
   END_RUNG
   RUNG wire#powerrail
      Contact( "BA040AZSSP201.00" )
      Contact( "Unit1.ControlNodes".AutoStartEnable )
      { S7_Templates := "time_type := Time" } #statTonTime[1].TON(pt := T#3s, et =>)
      Coil( "Unit1.EmNodes".stateCommandsExecute )
   END_RUNG
   // the same network as SCL:
   #statLocalInterface.modeRequests.production := "Safety.DataFromSafety".mainOp.auto AND NOT #statNoModeCmd AND NOT "Unit1.EmNodes".WakeupRecoveryRequired;
   #statLocalInterface.modeRequests.maintenance := "Safety.DataFromSafety".mainOp.manual AND "Safety.DataFromSafety".scsMode.setup AND #globalStatus.clock.cycle100Msec AND NOT #statNoModeCmd AND NOT "Unit1.EmNodes".WakeupRecoveryRequired;
   #statLocalInterface.modeRequests.manual := "Safety.DataFromSafety".mainOp.manual AND "Safety.DataFromSafety".scsMode.auto AND #globalStatus.clock.cycle100Msec AND NOT #statNoModeCmd AND NOT "Unit1.EmNodes".WakeupRecoveryRequired;
   #statTonTime[0].TON(IN := NOT (NOT "Safety.DataFromSafety".scsMode.disable AND "Safety.DataFromSafety".devicesSummary.allEstopButtonsOK AND NOT "Safety.DataFromSafety".BA60LightCurtainDetect) OR ("Safety.DataFromSafety".AllSFDoorOpen AND (NOT "Safety.DataFromSafety".rcMode1.RollChange OR NOT "Safety.DataFromSafety".statusZone2.SFDoorOpen) AND (NOT "Safety.DataFromSafety".rcMode2.RollChange OR NOT "Safety.DataFromSafety".statusZone3.SFDoorOpen) AND NOT "Safety.DataToSafety".MobilePanelConnected AND #FALSE) OR (NOT "Safety.DataFromSafety".AllSFDoorOpen AND "Safety.DataFromSafety".devicesSummary.anyDoorOpen) OR "Safety.DataFromSafety".SetupModFault,
                       PT := T#200ms);
   #statNoModeCmd := #statTonTime[0].Q;
   #statLocalInterface.modeRequests.nomode := #statNoModeCmd AND #globalStatus.clock.cycle100Msec AND NOT "Unit1.EmNodes".unitStatus.mode.nomode;
   #statLocalInterface.modeRequests.sleep := "Unit1.EmNodes".SleepModeChangeReq AND #globalStatus.clock.cycle100Msec;
   #statLocalInterface.modeRequests.deepsleep := "Unit1.EmNodes".DeepSleepModeChangeReq AND #globalStatus.clock.cycle100Msec;
   #statLocalInterface.stateCommands.reset := NOT (NOT "Safety.DataFromSafety".mainOp.reset AND NOT "Unit1.EmNodes".pHmiMode.reset) AND NOT "Unit1.EmNodes".unitStatus.state.aborted;
   #_w1 := "Safety.DataFromSafety".mainOp.home AND NOT #statPulse[0];   // rising edge of "Safety.DataFromSafety".mainOp.home
   #statPulse[0] := "Safety.DataFromSafety".mainOp.home;
   #statLocalInterface.stateCommands.start := ((#_w1 AND "Unit1.ControlNodes".InitializeEnable) OR #statLocalInterface.stateCommands.start) AND NOT "Unit1.EmNodes".unitStatus.state.starting;
   #_w2 := "Safety.DataFromSafety".BA10.Normalinterlocks.SCS_DisableMode AND NOT #statPulse[1];   // rising edge of "Safety.DataFromSafety".BA10.Normalinterlocks.SCS_DisableMode
   #statPulse[1] := "Safety.DataFromSafety".BA10.Normalinterlocks.SCS_DisableMode;
   #_w3 := "Safety.DataFromSafety".BA15.Normalinterlocks.SCS_DisableMode AND NOT #statPulse[2];   // rising edge of "Safety.DataFromSafety".BA15.Normalinterlocks.SCS_DisableMode
   #statPulse[2] := "Safety.DataFromSafety".BA15.Normalinterlocks.SCS_DisableMode;
   #_w4 := "Safety.DataFromSafety".BA60.Normalinterlocks.SCS_DisableMode AND NOT #statPulse[3];   // rising edge of "Safety.DataFromSafety".BA60.Normalinterlocks.SCS_DisableMode
   #statPulse[3] := "Safety.DataFromSafety".BA60.Normalinterlocks.SCS_DisableMode;
   #_w5 := "Safety.DataFromSafety".BA30.Normalinterlocks.SCS_DisableMode AND NOT #statPulse[4];   // rising edge of "Safety.DataFromSafety".BA30.Normalinterlocks.SCS_DisableMode
   #statPulse[4] := "Safety.DataFromSafety".BA30.Normalinterlocks.SCS_DisableMode;
   #statLocalInterface.stateCommands.stop := "BA040AZSSP201.01" OR NOT ("Safety.DataFromSafety".fDoorDrive.fDoor1.released AND "Safety.DataFromSafety".fDoorDrive.fDoor2.released AND "Safety.DataFromSafety".fDoorDrive.fDoor5.released AND "Safety.DataFromSafety".fDoorDrive.fDoor6.released AND "Safety.DataFromSafety".fDoorDrive.fDoor7.released AND "Safety.DataFromSafety".fDoorDrive.fDoor8.released AND "Safety.DataFromSafety".fDoorDrive.fDoor9.released AND "Safety.DataFromSafety".fDoorDrive.fDoor10.released) OR (NOT "Safety.DataFromSafety".fDoorDrive.fDoor3.released AND (NOT "Safety.DataFromSafety".rcMode1.RollChange OR NOT "Safety.DataFromSafety".scsMode.auto)) OR (NOT "Safety.DataFromSafety".fDoorDrive.fDoor4.released AND (NOT "Safety.DataFromSafety".rcMode2.RollChange OR NOT "Safety.DataFromSafety".scsMode.auto)) OR ((NOT (NOT "Safety.DataFromSafety".mainOp.manual AND NOT "Safety.DataFromSafety".scsMode.setup AND NOT "Safety.DataFromSafety".scsMode.disable) OR NOT (NOT "Safety.DataFromSafety".zone1DoorOpenRequest AND NOT "Safety.DataFromSafety".zone2DoorOpenRequest AND NOT "Safety.DataFromSafety".zone3DoorOpenRequest)) AND NOT "Unit1.EmNodes".unitStatus.simulationActive AND "Unit1.EmNodes".unitStatus.state.execute) OR ((#_w2 OR #_w3 OR #_w4 OR #_w5) AND #TRUE);
   #statLocalInterface.stateCommands.hold := #FALSE;
   #statLocalInterface.stateCommands.unhold := #FALSE;
   #statLocalInterface.stateCommands.suspend := (NOT "Unit1.EmNodes".unitStatus.specialFunctions.ReelCutCathodeUnuse AND "Unit1.EmNodes".BA010.ReelCutToStack.UnitStatus.commands.suspend) OR (NOT "Unit1.EmNodes".unitStatus.specialFunctions.ReelCutAnodeUnuse AND "Unit1.EmNodes".BA015.ReelCutToStack.UnitStatus.commands.suspend) OR (NOT "Unit1.EmNodes".unitStatus.specialFunctions.InspectionUnuse AND "Unit1.EmNodes".BA060.InspectionToStack.UnitStatus.commands.suspend);
   #statLocalInterface.stateCommands.unsuspend := (NOT "Unit1.EmNodes".unitStatus.specialFunctions.ReelCutCathodeUnuse AND "Unit1.EmNodes".BA010.ReelCutToStack.UnitStatus.commands.unsuspend) OR (NOT "Unit1.EmNodes".unitStatus.specialFunctions.ReelCutAnodeUnuse AND "Unit1.EmNodes".BA015.ReelCutToStack.UnitStatus.commands.unsuspend) OR (NOT "Unit1.EmNodes".unitStatus.specialFunctions.InspectionUnuse AND "Unit1.EmNodes".BA060.InspectionToStack.UnitStatus.commands.unsuspend);
   #statLocalInterface.stateCommands.abort := #FALSE;
   #statLocalInterface.stateCommands.clear := NOT (NOT "Safety.DataFromSafety".mainOp.reset AND NOT "Unit1.EmNodes".pHmiMode.reset) AND "Unit1.EmNodes".unitStatus.state.aborted AND #safetyReleased;
   #statLocalInterface.stateCommands.complete := "Unit1.EmData".RunOutModeControl.RunOutStart OR "Unit1.EmNodes".CapabilityModeComplete;
   #statLocalInterface.stateCommands.stateComplete := NOT (NOT "Unit1.EmNodes".unitStatus.state.aborting AND NOT "Unit1.EmNodes".unitStatus.state.clearing) AND #tempProcessCommands.stateComplete;
   #statTonTime[1].TON(IN := "BA040AZSSP201.00" AND "Unit1.ControlNodes".AutoStartEnable, PT := T#3s);
   "Unit1.EmNodes".stateCommandsExecute := #statTonTime[1].Q;
END_REGION

REGION Network 39: Main Op Lamp 수정
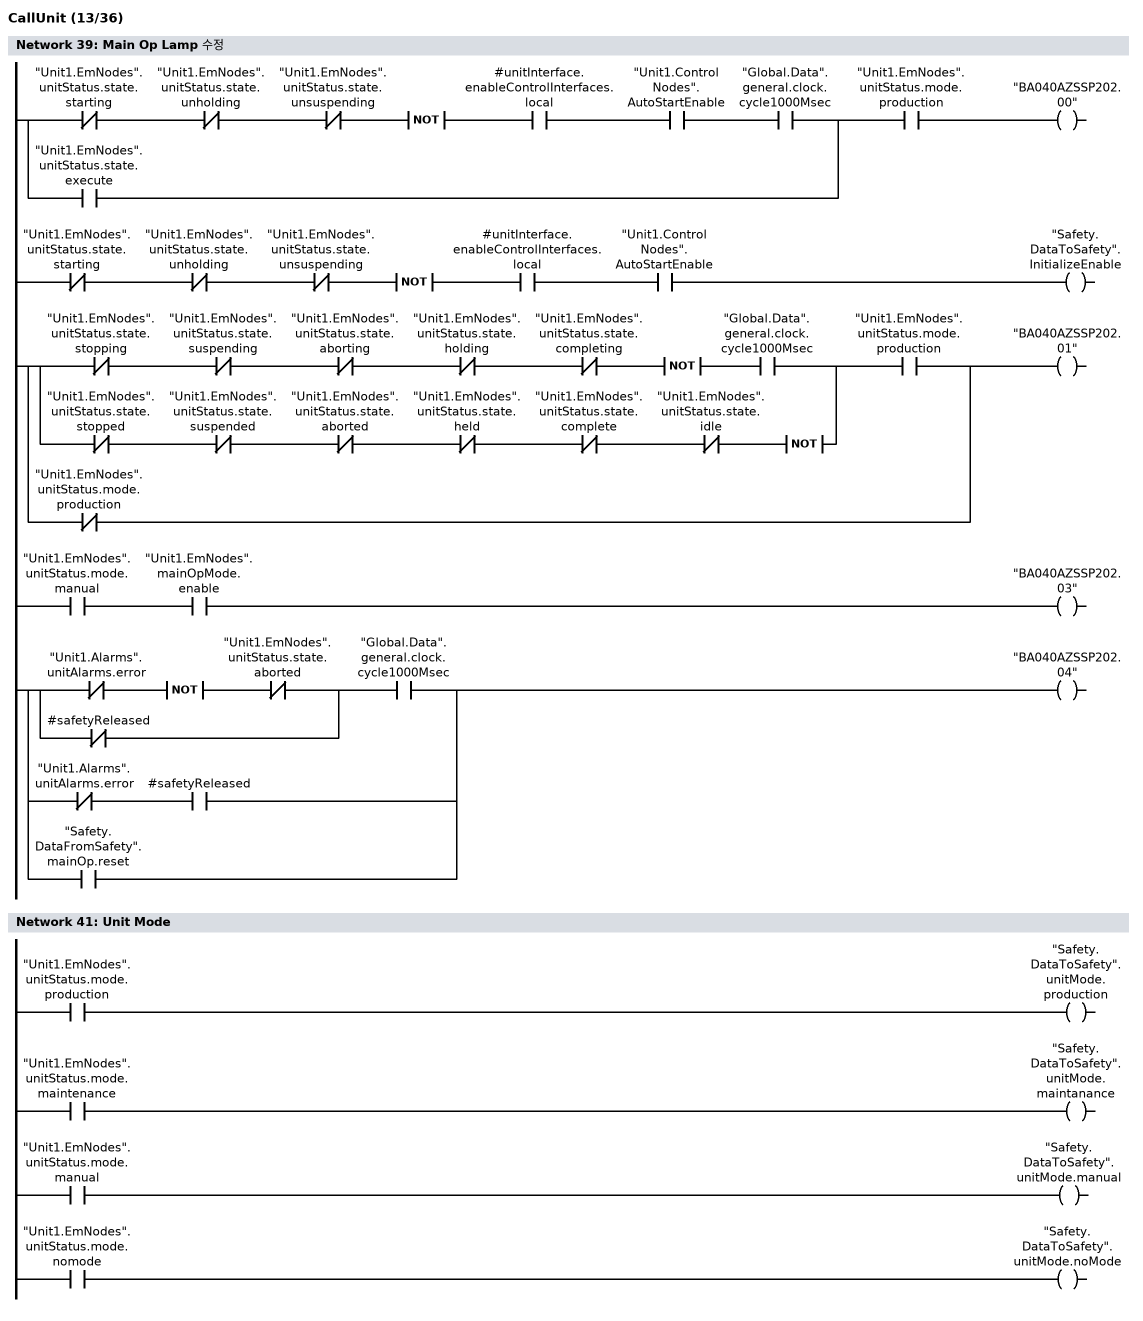
   RUNG wire#powerrail
      I_Contact( "Unit1.EmNodes".unitStatus.state.starting )
      I_Contact( "Unit1.EmNodes".unitStatus.state.unholding )
      I_Contact( "Unit1.EmNodes".unitStatus.state.unsuspending )
      Not()
      Contact( #unitInterface.enableControlInterfaces.local )
      Contact( "Unit1.ControlNodes".AutoStartEnable )
      Contact( "Global.Data".general.clock.cycle1000Msec )
      wire#w1
      Contact( "Unit1.EmNodes".unitStatus.mode.production )
      Coil( "BA040AZSSP202.00" )
   END_RUNG
   RUNG wire#powerrail
      Contact( "Unit1.EmNodes".unitStatus.state.execute )
   END_RUNG wire#w1
   RUNG wire#powerrail
      I_Contact( "Unit1.EmNodes".unitStatus.state.starting )
      I_Contact( "Unit1.EmNodes".unitStatus.state.unholding )
      I_Contact( "Unit1.EmNodes".unitStatus.state.unsuspending )
      Not()
      Contact( #unitInterface.enableControlInterfaces.local )
      Contact( "Unit1.ControlNodes".AutoStartEnable )
      Coil( "Safety.DataToSafety".InitializeEnable )
   END_RUNG
   RUNG wire#powerrail
      I_Contact( "Unit1.EmNodes".unitStatus.state.stopping )
      I_Contact( "Unit1.EmNodes".unitStatus.state.suspending )
      I_Contact( "Unit1.EmNodes".unitStatus.state.aborting )
      I_Contact( "Unit1.EmNodes".unitStatus.state.holding )
      I_Contact( "Unit1.EmNodes".unitStatus.state.completing )
      Not()
      Contact( "Global.Data".general.clock.cycle1000Msec )
      wire#w2
      Contact( "Unit1.EmNodes".unitStatus.mode.production )
      wire#w3
      Coil( "BA040AZSSP202.01" )
   END_RUNG
   RUNG wire#powerrail
      I_Contact( "Unit1.EmNodes".unitStatus.state.stopped )
      I_Contact( "Unit1.EmNodes".unitStatus.state.suspended )
      I_Contact( "Unit1.EmNodes".unitStatus.state.aborted )
      I_Contact( "Unit1.EmNodes".unitStatus.state.held )
      I_Contact( "Unit1.EmNodes".unitStatus.state.complete )
      I_Contact( "Unit1.EmNodes".unitStatus.state.idle )
      Not()
   END_RUNG wire#w2
   RUNG wire#powerrail
      I_Contact( "Unit1.EmNodes".unitStatus.mode.production )
   END_RUNG wire#w3
   RUNG wire#powerrail
      Contact( "Unit1.EmNodes".unitStatus.mode.manual )
      Contact( "Unit1.EmNodes".mainOpMode.enable )
      Coil( "BA040AZSSP202.03" )
   END_RUNG
   RUNG wire#powerrail
      I_Contact( "Unit1.Alarms".unitAlarms.error )
      Not()
      I_Contact( "Unit1.EmNodes".unitStatus.state.aborted )
      wire#w4
      Contact( "Global.Data".general.clock.cycle1000Msec )
      wire#w5
      Coil( "BA040AZSSP202.04" )
   END_RUNG
   RUNG wire#powerrail
      I_Contact( #safetyReleased )
   END_RUNG wire#w4
   RUNG wire#powerrail
      I_Contact( "Unit1.Alarms".unitAlarms.error )
      Contact( #safetyReleased )
   END_RUNG wire#w5
   RUNG wire#powerrail
      Contact( "Safety.DataFromSafety".mainOp.reset )
   END_RUNG wire#w5
   // the same network as SCL:
   "BA040AZSSP202.00" := ((NOT (NOT "Unit1.EmNodes".unitStatus.state.starting AND NOT "Unit1.EmNodes".unitStatus.state.unholding AND NOT "Unit1.EmNodes".unitStatus.state.unsuspending) AND #unitInterface.enableControlInterfaces.local AND "Unit1.ControlNodes".AutoStartEnable AND "Global.Data".general.clock.cycle1000Msec) OR "Unit1.EmNodes".unitStatus.state.execute) AND "Unit1.EmNodes".unitStatus.mode.production;
   "Safety.DataToSafety".InitializeEnable := NOT (NOT "Unit1.EmNodes".unitStatus.state.starting AND NOT "Unit1.EmNodes".unitStatus.state.unholding AND NOT "Unit1.EmNodes".unitStatus.state.unsuspending) AND #unitInterface.enableControlInterfaces.local AND "Unit1.ControlNodes".AutoStartEnable;
   "BA040AZSSP202.01" := (((NOT (NOT "Unit1.EmNodes".unitStatus.state.stopping AND NOT "Unit1.EmNodes".unitStatus.state.suspending AND NOT "Unit1.EmNodes".unitStatus.state.aborting AND NOT "Unit1.EmNodes".unitStatus.state.holding AND NOT "Unit1.EmNodes".unitStatus.state.completing) AND "Global.Data".general.clock.cycle1000Msec) OR NOT (NOT "Unit1.EmNodes".unitStatus.state.stopped AND NOT "Unit1.EmNodes".unitStatus.state.suspended AND NOT "Unit1.EmNodes".unitStatus.state.aborted AND NOT "Unit1.EmNodes".unitStatus.state.held AND NOT "Unit1.EmNodes".unitStatus.state.complete AND NOT "Unit1.EmNodes".unitStatus.state.idle)) AND "Unit1.EmNodes".unitStatus.mode.production) OR NOT "Unit1.EmNodes".unitStatus.mode.production;
   "BA040AZSSP202.03" := "Unit1.EmNodes".unitStatus.mode.manual AND "Unit1.EmNodes".mainOpMode.enable;
   "BA040AZSSP202.04" := (((NOT (NOT "Unit1.Alarms".unitAlarms.error) AND NOT "Unit1.EmNodes".unitStatus.state.aborted) OR NOT #safetyReleased) AND "Global.Data".general.clock.cycle1000Msec) OR (NOT "Unit1.Alarms".unitAlarms.error AND #safetyReleased) OR "Safety.DataFromSafety".mainOp.reset;
END_REGION

REGION Network 40: ******************** Data To Safety Mapping ********************
END_REGION

REGION Network 41: Unit Mode
   RUNG wire#powerrail
      Contact( "Unit1.EmNodes".unitStatus.mode.production )
      Coil( "Safety.DataToSafety".unitMode.production )
   END_RUNG
   RUNG wire#powerrail
      Contact( "Unit1.EmNodes".unitStatus.mode.maintenance )
      Coil( "Safety.DataToSafety".unitMode.maintanance )
   END_RUNG
   RUNG wire#powerrail
      Contact( "Unit1.EmNodes".unitStatus.mode.manual )
      Coil( "Safety.DataToSafety".unitMode.manual )
   END_RUNG
   RUNG wire#powerrail
      Contact( "Unit1.EmNodes".unitStatus.mode.nomode )
      Coil( "Safety.DataToSafety".unitMode.noMode )
   END_RUNG
   // the same network as SCL:
   "Safety.DataToSafety".unitMode.production := "Unit1.EmNodes".unitStatus.mode.production;
   "Safety.DataToSafety".unitMode.maintanance := "Unit1.EmNodes".unitStatus.mode.maintenance;
   "Safety.DataToSafety".unitMode.manual := "Unit1.EmNodes".unitStatus.mode.manual;
   "Safety.DataToSafety".unitMode.noMode := "Unit1.EmNodes".unitStatus.mode.nomode;
END_REGION

REGION Network 42: Unit States
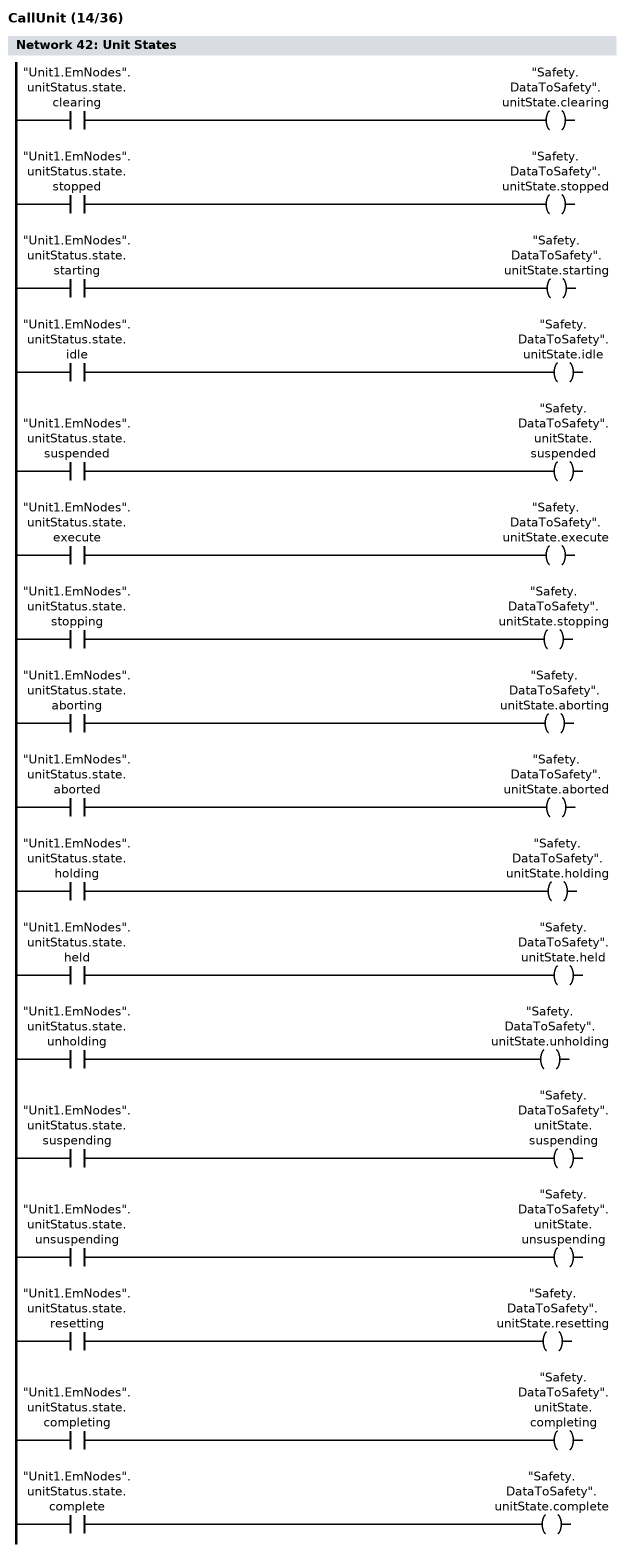
   RUNG wire#powerrail
      Contact( "Unit1.EmNodes".unitStatus.state.clearing )
      Coil( "Safety.DataToSafety".unitState.clearing )
   END_RUNG
   RUNG wire#powerrail
      Contact( "Unit1.EmNodes".unitStatus.state.stopped )
      Coil( "Safety.DataToSafety".unitState.stopped )
   END_RUNG
   RUNG wire#powerrail
      Contact( "Unit1.EmNodes".unitStatus.state.starting )
      Coil( "Safety.DataToSafety".unitState.starting )
   END_RUNG
   RUNG wire#powerrail
      Contact( "Unit1.EmNodes".unitStatus.state.idle )
      Coil( "Safety.DataToSafety".unitState.idle )
   END_RUNG
   RUNG wire#powerrail
      Contact( "Unit1.EmNodes".unitStatus.state.suspended )
      Coil( "Safety.DataToSafety".unitState.suspended )
   END_RUNG
   RUNG wire#powerrail
      Contact( "Unit1.EmNodes".unitStatus.state.execute )
      Coil( "Safety.DataToSafety".unitState.execute )
   END_RUNG
   RUNG wire#powerrail
      Contact( "Unit1.EmNodes".unitStatus.state.stopping )
      Coil( "Safety.DataToSafety".unitState.stopping )
   END_RUNG
   RUNG wire#powerrail
      Contact( "Unit1.EmNodes".unitStatus.state.aborting )
      Coil( "Safety.DataToSafety".unitState.aborting )
   END_RUNG
   RUNG wire#powerrail
      Contact( "Unit1.EmNodes".unitStatus.state.aborted )
      Coil( "Safety.DataToSafety".unitState.aborted )
   END_RUNG
   RUNG wire#powerrail
      Contact( "Unit1.EmNodes".unitStatus.state.holding )
      Coil( "Safety.DataToSafety".unitState.holding )
   END_RUNG
   RUNG wire#powerrail
      Contact( "Unit1.EmNodes".unitStatus.state.held )
      Coil( "Safety.DataToSafety".unitState.held )
   END_RUNG
   RUNG wire#powerrail
      Contact( "Unit1.EmNodes".unitStatus.state.unholding )
      Coil( "Safety.DataToSafety".unitState.unholding )
   END_RUNG
   RUNG wire#powerrail
      Contact( "Unit1.EmNodes".unitStatus.state.suspending )
      Coil( "Safety.DataToSafety".unitState.suspending )
   END_RUNG
   RUNG wire#powerrail
      Contact( "Unit1.EmNodes".unitStatus.state.unsuspending )
      Coil( "Safety.DataToSafety".unitState.unsuspending )
   END_RUNG
   RUNG wire#powerrail
      Contact( "Unit1.EmNodes".unitStatus.state.resetting )
      Coil( "Safety.DataToSafety".unitState.resetting )
   END_RUNG
   RUNG wire#powerrail
      Contact( "Unit1.EmNodes".unitStatus.state.completing )
      Coil( "Safety.DataToSafety".unitState.completing )
   END_RUNG
   RUNG wire#powerrail
      Contact( "Unit1.EmNodes".unitStatus.state.complete )
      Coil( "Safety.DataToSafety".unitState.complete )
   END_RUNG
   // the same network as SCL:
   "Safety.DataToSafety".unitState.clearing := "Unit1.EmNodes".unitStatus.state.clearing;
   "Safety.DataToSafety".unitState.stopped := "Unit1.EmNodes".unitStatus.state.stopped;
   "Safety.DataToSafety".unitState.starting := "Unit1.EmNodes".unitStatus.state.starting;
   "Safety.DataToSafety".unitState.idle := "Unit1.EmNodes".unitStatus.state.idle;
   "Safety.DataToSafety".unitState.suspended := "Unit1.EmNodes".unitStatus.state.suspended;
   "Safety.DataToSafety".unitState.execute := "Unit1.EmNodes".unitStatus.state.execute;
   "Safety.DataToSafety".unitState.stopping := "Unit1.EmNodes".unitStatus.state.stopping;
   "Safety.DataToSafety".unitState.aborting := "Unit1.EmNodes".unitStatus.state.aborting;
   "Safety.DataToSafety".unitState.aborted := "Unit1.EmNodes".unitStatus.state.aborted;
   "Safety.DataToSafety".unitState.holding := "Unit1.EmNodes".unitStatus.state.holding;
   "Safety.DataToSafety".unitState.held := "Unit1.EmNodes".unitStatus.state.held;
   "Safety.DataToSafety".unitState.unholding := "Unit1.EmNodes".unitStatus.state.unholding;
   "Safety.DataToSafety".unitState.suspending := "Unit1.EmNodes".unitStatus.state.suspending;
   "Safety.DataToSafety".unitState.unsuspending := "Unit1.EmNodes".unitStatus.state.unsuspending;
   "Safety.DataToSafety".unitState.resetting := "Unit1.EmNodes".unitStatus.state.resetting;
   "Safety.DataToSafety".unitState.completing := "Unit1.EmNodes".unitStatus.state.completing;
   "Safety.DataToSafety".unitState.complete := "Unit1.EmNodes".unitStatus.state.complete;
END_REGION

REGION Network 43: Deselect BA10, BA15, BA60
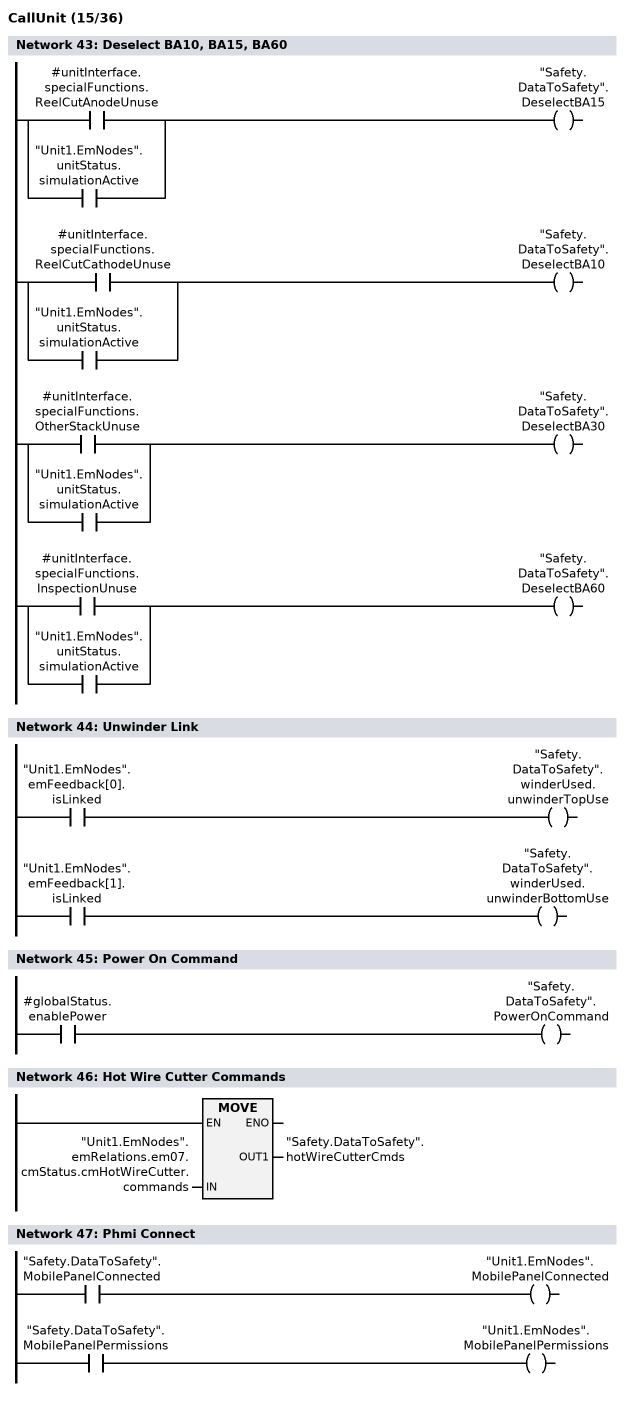
   RUNG wire#powerrail
      Contact( #unitInterface.specialFunctions.ReelCutAnodeUnuse )
      wire#w1
      Coil( "Safety.DataToSafety".DeselectBA15 )
   END_RUNG
   RUNG wire#powerrail
      Contact( "Unit1.EmNodes".unitStatus.simulationActive )
   END_RUNG wire#w1
   RUNG wire#powerrail
      Contact( #unitInterface.specialFunctions.ReelCutCathodeUnuse )
      wire#w2
      Coil( "Safety.DataToSafety".DeselectBA10 )
   END_RUNG
   RUNG wire#powerrail
      Contact( "Unit1.EmNodes".unitStatus.simulationActive )
   END_RUNG wire#w2
   RUNG wire#powerrail
      Contact( #unitInterface.specialFunctions.OtherStackUnuse )
      wire#w3
      Coil( "Safety.DataToSafety".DeselectBA30 )
   END_RUNG
   RUNG wire#powerrail
      Contact( "Unit1.EmNodes".unitStatus.simulationActive )
   END_RUNG wire#w3
   RUNG wire#powerrail
      Contact( #unitInterface.specialFunctions.InspectionUnuse )
      wire#w4
      Coil( "Safety.DataToSafety".DeselectBA60 )
   END_RUNG
   RUNG wire#powerrail
      Contact( "Unit1.EmNodes".unitStatus.simulationActive )
   END_RUNG wire#w4
   // the same network as SCL:
   "Safety.DataToSafety".DeselectBA15 := #unitInterface.specialFunctions.ReelCutAnodeUnuse OR "Unit1.EmNodes".unitStatus.simulationActive;
   "Safety.DataToSafety".DeselectBA10 := #unitInterface.specialFunctions.ReelCutCathodeUnuse OR "Unit1.EmNodes".unitStatus.simulationActive;
   "Safety.DataToSafety".DeselectBA30 := #unitInterface.specialFunctions.OtherStackUnuse OR "Unit1.EmNodes".unitStatus.simulationActive;
   "Safety.DataToSafety".DeselectBA60 := #unitInterface.specialFunctions.InspectionUnuse OR "Unit1.EmNodes".unitStatus.simulationActive;
END_REGION

REGION Network 44: Unwinder Link
   RUNG wire#powerrail
      Contact( "Unit1.EmNodes".emFeedback[0].isLinked )
      Coil( "Safety.DataToSafety".winderUsed.unwinderTopUse )
   END_RUNG
   RUNG wire#powerrail
      Contact( "Unit1.EmNodes".emFeedback[1].isLinked )
      Coil( "Safety.DataToSafety".winderUsed.unwinderBottomUse )
   END_RUNG
   // the same network as SCL:
   "Safety.DataToSafety".winderUsed.unwinderTopUse := "Unit1.EmNodes".emFeedback[0].isLinked;
   "Safety.DataToSafety".winderUsed.unwinderBottomUse := "Unit1.EmNodes".emFeedback[1].isLinked;
END_REGION

REGION Network 45: Power On Command
   RUNG wire#powerrail
      Contact( #globalStatus.enablePower )
      Coil( "Safety.DataToSafety".PowerOnCommand )
   END_RUNG
   // the same network as SCL:
   "Safety.DataToSafety".PowerOnCommand := #globalStatus.enablePower;
END_REGION

REGION Network 46: Hot Wire Cutter Commands
   RUNG wire#powerrail
      Move(in := "Unit1.EmNodes".emRelations.em07.cmStatus.cmHotWireCutter.commands, out1 => "Safety.DataToSafety".hotWireCutterCmds)
   END_RUNG
   // the same network as SCL:
   "Safety.DataToSafety".hotWireCutterCmds := "Unit1.EmNodes".emRelations.em07.cmStatus.cmHotWireCutter.commands;
END_REGION

REGION Network 47: Phmi Connect
   RUNG wire#powerrail
      Contact( "Safety.DataToSafety".MobilePanelConnected )
      Coil( "Unit1.EmNodes".MobilePanelConnected )
   END_RUNG
   RUNG wire#powerrail
      Contact( "Safety.DataToSafety".MobilePanelPermissions )
      Coil( "Unit1.EmNodes".MobilePanelPermissions )
   END_RUNG
   // the same network as SCL:
   "Unit1.EmNodes".MobilePanelConnected := "Safety.DataToSafety".MobilePanelConnected;
   "Unit1.EmNodes".MobilePanelPermissions := "Safety.DataToSafety".MobilePanelPermissions;
END_REGION

REGION Network 48: SepaGripper Axis Move To BA60
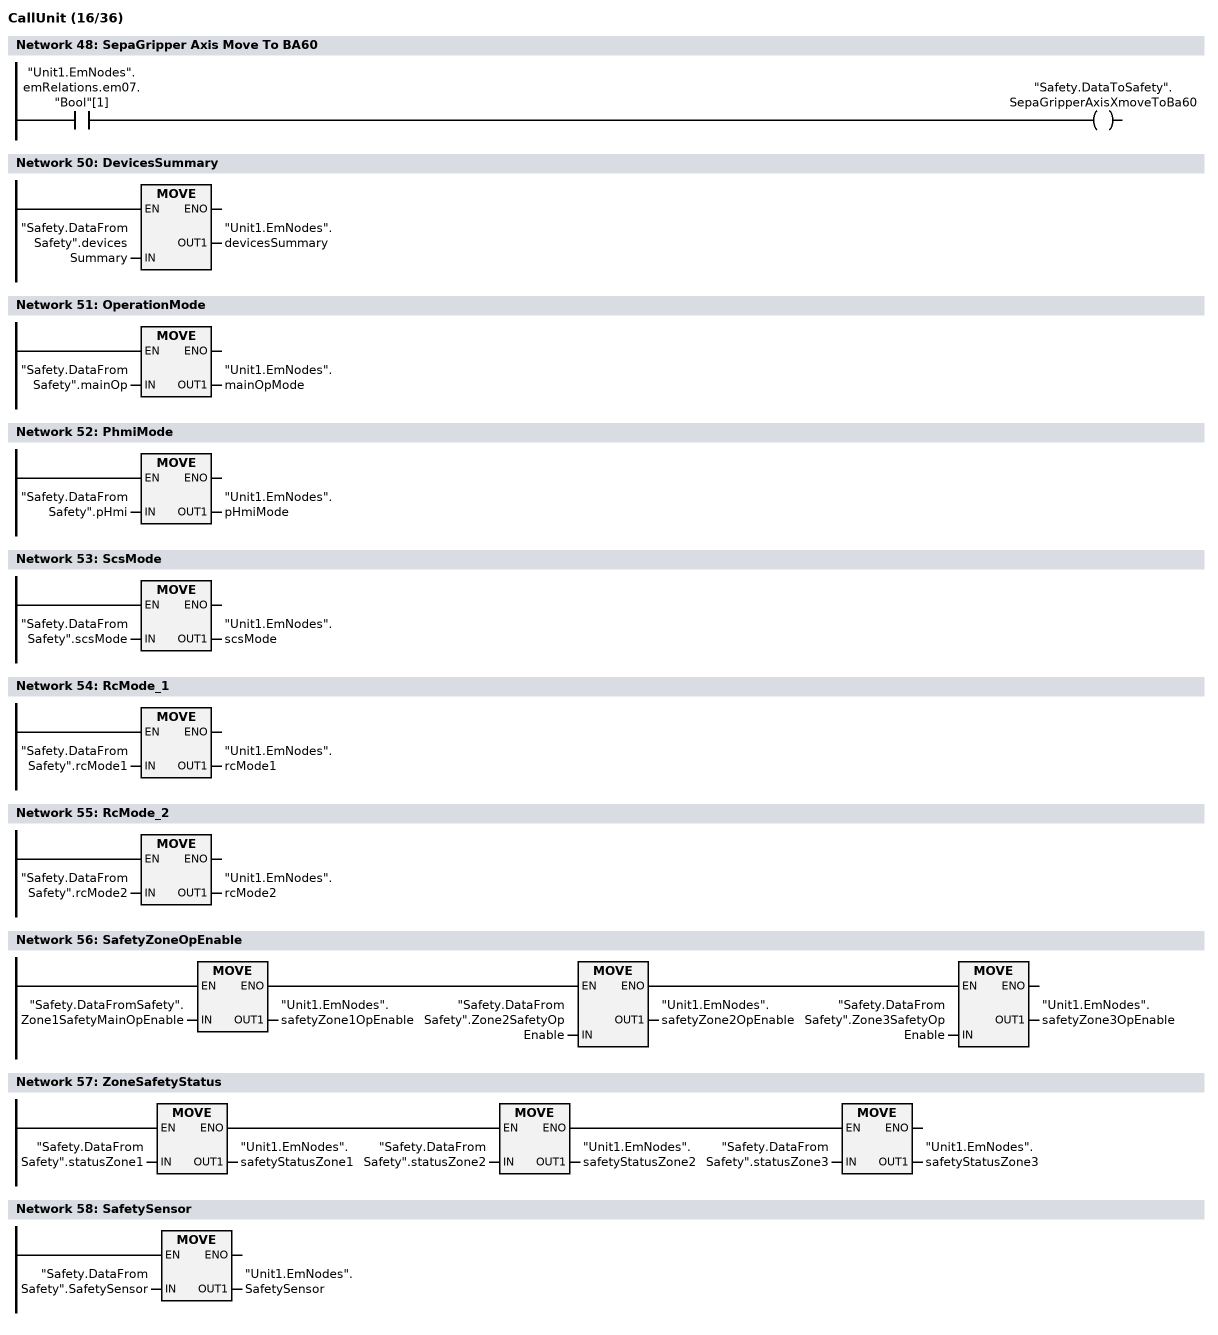
   RUNG wire#powerrail
      Contact( "Unit1.EmNodes".emRelations.em07."Bool"[1] )
      Coil( "Safety.DataToSafety".SepaGripperAxisXmoveToBa60 )
   END_RUNG
   // the same network as SCL:
   "Safety.DataToSafety".SepaGripperAxisXmoveToBa60 := "Unit1.EmNodes".emRelations.em07."Bool"[1];
END_REGION

REGION Network 49: ******************** Data From Safety Mapping ********************
END_REGION

REGION Network 50: DevicesSummary
   RUNG wire#powerrail
      Move(in := "Safety.DataFromSafety".devicesSummary, out1 => "Unit1.EmNodes".devicesSummary)
   END_RUNG
   // the same network as SCL:
   "Unit1.EmNodes".devicesSummary := "Safety.DataFromSafety".devicesSummary;
END_REGION

REGION Network 51: OperationMode
   RUNG wire#powerrail
      Move(in := "Safety.DataFromSafety".mainOp, out1 => "Unit1.EmNodes".mainOpMode)
   END_RUNG
   // the same network as SCL:
   "Unit1.EmNodes".mainOpMode := "Safety.DataFromSafety".mainOp;
END_REGION

REGION Network 52: PhmiMode
   RUNG wire#powerrail
      Move(in := "Safety.DataFromSafety".pHmi, out1 => "Unit1.EmNodes".pHmiMode)
   END_RUNG
   // the same network as SCL:
   "Unit1.EmNodes".pHmiMode := "Safety.DataFromSafety".pHmi;
END_REGION

